LIN {X 103.742,Y 102.138,Z 83.038,A 180.000,B 0.000,C 180.000} C_DIS
LIN {X 103.836,Y 102.012,Z 83.035,A 180.000,B 0.000,C 180.000} C_DIS
LIN {X 103.928,Y 101.885,Z 83.032,A 180.000,B 0.000,C 180.000} C_DIS
LIN {X 104.017,Y 101.755,Z 83.030,A 180.000,B 0.000,C 180.000} C_DIS
LIN {X 104.184,Y 101.489,Z 83.025,A 180.000,B 0.000,C 180.000} C_DIS
LIN {X 104.341,Y 101.216,Z 83.021,A 180.000,B 0.000,C 180.000} C_DIS
LIN {X 104.489,Y 100.938,Z 83.017,A 180.000,B 0.000,C 180.000} C_DIS
LIN {X 104.623,Y 100.654,Z 83.013,A 180.000,B 0.000,C 180.000} C_DIS
LIN {X 104.744,Y 100.363,Z 83.010,A 180.000,B 0.000,C 180.000} C_DIS
LIN {X 104.858,Y 100.069,Z 83.007,A 180.000,B 0.000,C 180.000} C_DIS
LIN {X 104.957,Y 99.770,Z 83.005,A 180.000,B 0.000,C 180.000} C_DIS
LIN {X 105.040,Y 99.466,Z 83.003,A 180.000,B 0.000,C 180.000} C_DIS
LIN {X 105.117,Y 99.161,Z 83.001,A 180.000,B 0.000,C 180.000} C_DIS
LIN {X 105.179,Y 98.852,Z 83.000,A 180.000,B 0.000,C 180.000} C_DIS
LIN {X 105.224,Y 98.540,Z 83.000,A 180.000,B 0.000,C 180.000} C_DIS
LIN {X 105.239,Y 98.417,Z 83.000,A 180.000,B 0.000,C 180.000} C_DIS
; Cutting Move Starts
LIN {X 105.250,Y 98.327,Z 83.000,A 180.000,B 0.000,C 180.000} C_DIS
LIN {X 105.268,Y 98.148,Z 83.000,A 180.000,B 0.000,C 180.000} C_DIS
LIN {X 105.282,Y 97.969,Z 83.000,A 180.000,B 0.000,C 180.000} C_DIS
LIN {X 105.289,Y 97.790,Z 83.000,A 180.000,B 0.000,C 180.000} C_DIS
LIN {X 105.293,Y 97.612,Z 83.000,A 180.000,B 0.000,C 180.000} C_DIS
LIN {X 105.293,Y 97.433,Z 83.000,A 180.000,B 0.000,C 180.000} C_DIS
LIN {X 105.290,Y 97.254,Z 83.000,A 180.000,B 0.000,C 180.000} C_DIS
LIN {X 105.285,Y 97.075,Z 83.000,A 180.000,B 0.000,C 180.000} C_DIS
LIN {X 105.272,Y 96.897,Z 83.000,A 180.000,B 0.000,C 180.000} C_DIS
LIN {X 105.256,Y 96.718,Z 83.000,A 180.000,B 0.000,C 180.000} C_DIS
LIN {X 105.233,Y 96.539,Z 83.000,A 180.000,B 0.000,C 180.000} C_DIS
LIN {X 105.210,Y 96.360,Z 83.000,A 180.000,B 0.000,C 180.000} C_DIS
LIN {X 105.184,Y 96.181,Z 83.000,A 180.000,B 0.000,C 180.000} C_DIS
LIN {X 105.150,Y 96.003,Z 83.000,A 180.000,B 0.000,C 180.000} C_DIS
LIN {X 105.120,Y 95.853,Z 83.000,A 180.000,B 0.000,C 180.000} C_DIS
LIN {X 105.113,Y 95.824,Z 83.000,A 180.000,B 0.000,C 180.000} C_DIS
LIN {X 105.068,Y 95.645,Z 83.000,A 180.000,B 0.000,C 180.000} C_DIS
LIN {X 105.022,Y 95.466,Z 83.000,A 180.000,B 0.000,C 180.000} C_DIS
LIN {X 104.975,Y 95.288,Z 83.000,A 180.000,B 0.000,C 180.000} C_DIS
LIN {X 104.941,Y 95.177,Z 83.000,A 180.000,B 0.000,C 180.000} C_DIS
LIN {X 104.920,Y 95.109,Z 83.000,A 180.000,B 0.000,C 180.000} C_DIS
LIN {X 104.860,Y 94.930,Z 83.000,A 180.000,B 0.000,C 180.000} C_DIS
LIN {X 104.792,Y 94.751,Z 83.000,A 180.000,B 0.000,C 180.000} C_DIS
LIN {X 104.762,Y 94.674,Z 83.000,A 180.000,B 0.000,C 180.000} C_DIS
LIN {X 104.722,Y 94.573,Z 83.000,A 180.000,B 0.000,C 180.000} C_DIS
LIN {X 104.650,Y 94.394,Z 83.000,A 180.000,B 0.000,C 180.000} C_DIS
LIN {X 104.584,Y 94.246,Z 83.000,A 180.000,B 0.000,C 180.000} C_DIS
LIN {X 104.570,Y 94.215,Z 83.000,A 180.000,B 0.000,C 180.000} C_DIS
LIN {X 104.483,Y 94.036,Z 83.000,A 180.000,B 0.000,C 180.000} C_DIS
LIN {X 104.405,Y 93.885,Z 83.000,A 180.000,B 0.000,C 180.000} C_DIS
LIN {X 104.391,Y 93.857,Z 83.000,A 180.000,B 0.000,C 180.000} C_DIS
LIN {X 104.292,Y 93.679,Z 83.000,A 180.000,B 0.000,C 180.000} C_DIS
LIN {X 104.226,Y 93.561,Z 83.000,A 180.000,B 0.000,C 180.000} C_DIS
LIN {X 104.190,Y 93.500,Z 83.000,A 180.000,B 0.000,C 180.000} C_DIS
LIN {X 104.082,Y 93.321,Z 83.000,A 180.000,B 0.000,C 180.000} C_DIS
LIN {X 104.047,Y 93.269,Z 83.000,A 180.000,B 0.000,C 180.000} C_DIS
LIN {X 103.963,Y 93.142,Z 83.000,A 180.000,B 0.000,C 180.000} C_DIS
LIN {X 103.869,Y 93.008,Z 83.000,A 180.000,B 0.000,C 180.000} C_DIS
LIN {X 103.837,Y 92.964,Z 83.000,A 180.000,B 0.000,C 180.000} C_DIS
LIN {X 103.705,Y 92.785,Z 83.000,A 180.000,B 0.000,C 180.000} C_DIS
LIN {X 103.690,Y 92.764,Z 83.000,A 180.000,B 0.000,C 180.000} C_DIS
LIN {X 103.569,Y 92.606,Z 83.000,A 180.000,B 0.000,C 180.000} C_DIS
LIN {X 103.511,Y 92.536,Z 83.000,A 180.000,B 0.000,C 180.000} C_DIS
LIN {X 103.419,Y 92.427,Z 83.000,A 180.000,B 0.000,C 180.000} C_DIS
LIN {X 103.332,Y 92.328,Z 83.000,A 180.000,B 0.000,C 180.000} C_DIS
LIN {X 103.258,Y 92.249,Z 83.000,A 180.000,B 0.000,C 180.000} C_DIS
LIN {X 103.153,Y 92.138,Z 83.000,A 180.000,B 0.000,C 180.000} C_DIS
LIN {X 103.089,Y 92.070,Z 83.000,A 180.000,B 0.000,C 180.000} C_DIS
LIN {X 102.975,Y 91.950,Z 83.000,A 180.000,B 0.000,C 180.000} C_DIS
LIN {X 102.914,Y 91.891,Z 83.000,A 180.000,B 0.000,C 180.000} C_DIS
LIN {X 102.796,Y 91.779,Z 83.000,A 180.000,B 0.000,C 180.000} C_DIS
LIN {X 102.723,Y 91.712,Z 83.000,A 180.000,B 0.000,C 180.000} C_DIS
LIN {X 102.617,Y 91.622,Z 83.000,A 180.000,B 0.000,C 180.000} C_DIS
LIN {X 102.513,Y 91.533,Z 83.000,A 180.000,B 0.000,C 180.000} C_DIS
LIN {X 102.438,Y 91.472,Z 83.000,A 180.000,B 0.000,C 180.000} C_DIS
LIN {X 102.296,Y 91.355,Z 83.000,A 180.000,B 0.000,C 180.000} C_DIS
LIN {X 102.260,Y 91.326,Z 83.000,A 180.000,B 0.000,C 180.000} C_DIS
LIN {X 102.081,Y 91.192,Z 83.000,A 180.000,B 0.000,C 180.000} C_DIS
LIN {X 102.060,Y 91.176,Z 83.000,A 180.000,B 0.000,C 180.000} C_DIS
LIN {X 101.902,Y 91.068,Z 83.000,A 180.000,B 0.000,C 180.000} C_DIS
LIN {X 101.796,Y 90.997,Z 83.000,A 180.000,B 0.000,C 180.000} C_DIS
LIN {X 101.723,Y 90.950,Z 83.000,A 180.000,B 0.000,C 180.000} C_DIS
LIN {X 101.545,Y 90.837,Z 83.000,A 180.000,B 0.000,C 180.000} C_DIS
LIN {X 101.514,Y 90.818,Z 83.000,A 180.000,B 0.000,C 180.000} C_DIS
LIN {X 101.366,Y 90.731,Z 83.000,A 180.000,B 0.000,C 180.000} C_DIS
LIN {X 101.203,Y 90.640,Z 83.000,A 180.000,B 0.000,C 180.000} C_DIS
LIN {X 101.187,Y 90.631,Z 83.000,A 180.000,B 0.000,C 180.000} C_DIS
LIN {X 101.008,Y 90.539,Z 83.000,A 180.000,B 0.000,C 180.000} C_DIS
LIN {X 100.844,Y 90.461,Z 83.000,A 180.000,B 0.000,C 180.000} C_DIS
LIN {X 100.829,Y 90.454,Z 83.000,A 180.000,B 0.000,C 180.000} C_DIS
LIN {X 100.651,Y 90.372,Z 83.000,A 180.000,B 0.000,C 180.000} C_DIS
LIN {X 100.472,Y 90.292,Z 83.000,A 180.000,B 0.000,C 180.000} C_DIS
LIN {X 100.447,Y 90.282,Z 83.000,A 180.000,B 0.000,C 180.000} C_DIS
LIN {X 100.293,Y 90.222,Z 83.000,A 180.000,B 0.000,C 180.000} C_DIS
LIN {X 100.114,Y 90.156,Z 83.000,A 180.000,B 0.000,C 180.000} C_DIS
LIN {X 99.951,Y 90.103,Z 83.000,A 180.000,B 0.000,C 180.000} C_DIS
LIN {X 99.936,Y 90.098,Z 83.000,A 180.000,B 0.000,C 180.000} C_DIS
LIN {X 99.757,Y 90.041,Z 83.000,A 180.000,B 0.000,C 180.000} C_DIS
LIN {X 99.578,Y 89.986,Z 83.000,A 180.000,B 0.000,C 180.000} C_DIS
LIN {X 99.399,Y 89.939,Z 83.000,A 180.000,B 0.000,C 180.000} C_DIS
LIN {X 99.341,Y 89.925,Z 83.000,A 180.000,B 0.000,C 180.000} C_DIS
LIN {X 99.221,Y 89.897,Z 83.000,A 180.000,B 0.000,C 180.000} C_DIS
LIN {X 99.042,Y 89.861,Z 83.000,A 180.000,B 0.000,C 180.000} C_DIS
LIN {X 98.863,Y 89.827,Z 83.000,A 180.000,B 0.000,C 180.000} C_DIS
LIN {X 98.684,Y 89.795,Z 83.000,A 180.000,B 0.000,C 180.000} C_DIS
LIN {X 98.505,Y 89.770,Z 83.000,A 180.000,B 0.000,C 180.000} C_DIS
LIN {X 98.327,Y 89.748,Z 83.000,A 180.000,B 0.000,C 180.000} C_DIS
LIN {X 98.148,Y 89.733,Z 83.000,A 180.000,B 0.000,C 180.000} C_DIS
LIN {X 97.969,Y 89.721,Z 83.000,A 180.000,B 0.000,C 180.000} C_DIS
LIN {X 97.790,Y 89.711,Z 83.000,A 180.000,B 0.000,C 180.000} C_DIS
LIN {X 97.612,Y 89.705,Z 83.000,A 180.000,B 0.000,C 180.000} C_DIS
LIN {X 97.433,Y 89.704,Z 83.000,A 180.000,B 0.000,C 180.000} C_DIS
LIN {X 97.254,Y 89.709,Z 83.000,A 180.000,B 0.000,C 180.000} C_DIS
LIN {X 97.075,Y 89.718,Z 83.000,A 180.000,B 0.000,C 180.000} C_DIS
LIN {X 96.897,Y 89.730,Z 83.000,A 180.000,B 0.000,C 180.000} C_DIS
LIN {X 96.718,Y 89.745,Z 83.000,A 180.000,B 0.000,C 180.000} C_DIS
LIN {X 96.704,Y 89.746,Z 83.000,A 180.000,B 0.000,C 180.000} C_DIS
LIN {X 96.539,Y 89.763,Z 83.000,A 180.000,B 0.000,C 180.000} C_DIS
LIN {X 96.360,Y 89.789,Z 83.000,A 180.000,B 0.000,C 180.000} C_DIS
LIN {X 96.181,Y 89.819,Z 83.000,A 180.000,B 0.000,C 180.000} C_DIS
LIN {X 96.003,Y 89.853,Z 83.000,A 180.000,B 0.000,C 180.000} C_DIS
LIN {X 95.824,Y 89.888,Z 83.000,A 180.000,B 0.000,C 180.000} C_DIS
LIN {X 95.659,Y 89.925,Z 83.000,A 180.000,B 0.000,C 180.000} C_DIS
LIN {X 95.645,Y 89.928,Z 83.000,A 180.000,B 0.000,C 180.000} C_DIS
LIN {X 95.466,Y 89.974,Z 83.000,A 180.000,B 0.000,C 180.000} C_DIS
LIN {X 95.288,Y 90.027,Z 83.000,A 180.000,B 0.000,C 180.000} C_DIS
LIN {X 95.109,Y 90.084,Z 83.000,A 180.000,B 0.000,C 180.000} C_DIS
LIN {X 94.930,Y 90.142,Z 83.000,A 180.000,B 0.000,C 180.000} C_DIS
LIN {X 94.751,Y 90.205,Z 83.000,A 180.000,B 0.000,C 180.000} C_DIS
LIN {X 94.573,Y 90.274,Z 83.000,A 180.000,B 0.000,C 180.000} C_DIS
LIN {X 94.553,Y 90.282,Z 83.000,A 180.000,B 0.000,C 180.000} C_DIS
LIN {X 94.394,Y 90.352,Z 83.000,A 180.000,B 0.000,C 180.000} C_DIS
LIN {X 94.215,Y 90.433,Z 83.000,A 180.000,B 0.000,C 180.000} C_DIS
LIN {X 94.156,Y 90.461,Z 83.000,A 180.000,B 0.000,C 180.000} C_DIS
LIN {X 94.036,Y 90.517,Z 83.000,A 180.000,B 0.000,C 180.000} C_DIS
LIN {X 93.857,Y 90.608,Z 83.000,A 180.000,B 0.000,C 180.000} C_DIS
LIN {X 93.797,Y 90.640,Z 83.000,A 180.000,B 0.000,C 180.000} C_DIS
LIN {X 93.679,Y 90.705,Z 83.000,A 180.000,B 0.000,C 180.000} C_DIS
LIN {X 93.500,Y 90.810,Z 83.000,A 180.000,B 0.000,C 180.000} C_DIS
LIN {X 93.486,Y 90.818,Z 83.000,A 180.000,B 0.000,C 180.000} C_DIS
LIN {X 93.321,Y 90.922,Z 83.000,A 180.000,B 0.000,C 180.000} C_DIS
LIN {X 93.204,Y 90.997,Z 83.000,A 180.000,B 0.000,C 180.000} C_DIS
LIN {X 93.142,Y 91.038,Z 83.000,A 180.000,B 0.000,C 180.000} C_DIS
LIN {X 92.964,Y 91.159,Z 83.000,A 180.000,B 0.000,C 180.000} C_DIS
LIN {X 92.940,Y 91.176,Z 83.000,A 180.000,B 0.000,C 180.000} C_DIS
LIN {X 92.785,Y 91.293,Z 83.000,A 180.000,B 0.000,C 180.000} C_DIS
LIN {X 92.704,Y 91.355,Z 83.000,A 180.000,B 0.000,C 180.000} C_DIS
LIN {X 92.606,Y 91.435,Z 83.000,A 180.000,B 0.000,C 180.000} C_DIS
LIN {X 92.487,Y 91.533,Z 83.000,A 180.000,B 0.000,C 180.000} C_DIS
LIN {X 92.427,Y 91.584,Z 83.000,A 180.000,B 0.000,C 180.000} C_DIS
LIN {X 92.277,Y 91.712,Z 83.000,A 180.000,B 0.000,C 180.000} C_DIS
LIN {X 92.249,Y 91.738,Z 83.000,A 180.000,B 0.000,C 180.000} C_DIS
LIN {X 92.086,Y 91.891,Z 83.000,A 180.000,B 0.000,C 180.000} C_DIS
LIN {X 92.070,Y 91.906,Z 83.000,A 180.000,B 0.000,C 180.000} C_DIS
LIN {X 91.911,Y 92.070,Z 83.000,A 180.000,B 0.000,C 180.000} C_DIS
LIN {X 91.891,Y 92.091,Z 83.000,A 180.000,B 0.000,C 180.000} C_DIS
LIN {X 91.742,Y 92.249,Z 83.000,A 180.000,B 0.000,C 180.000} C_DIS
LIN {X 91.712,Y 92.281,Z 83.000,A 180.000,B 0.000,C 180.000} C_DIS
LIN {X 91.581,Y 92.427,Z 83.000,A 180.000,B 0.000,C 180.000} C_DIS
LIN {X 91.533,Y 92.483,Z 83.000,A 180.000,B 0.000,C 180.000} C_DIS
LIN {X 91.431,Y 92.606,Z 83.000,A 180.000,B 0.000,C 180.000} C_DIS
LIN {X 91.355,Y 92.705,Z 83.000,A 180.000,B 0.000,C 180.000} C_DIS
LIN {X 91.295,Y 92.785,Z 83.000,A 180.000,B 0.000,C 180.000} C_DIS
LIN {X 91.176,Y 92.946,Z 83.000,A 180.000,B 0.000,C 180.000} C_DIS
LIN {X 91.163,Y 92.964,Z 83.000,A 180.000,B 0.000,C 180.000} C_DIS
LIN {X 91.037,Y 93.142,Z 83.000,A 180.000,B 0.000,C 180.000} C_DIS
LIN {X 90.997,Y 93.202,Z 83.000,A 180.000,B 0.000,C 180.000} C_DIS
LIN {X 90.918,Y 93.321,Z 83.000,A 180.000,B 0.000,C 180.000} C_DIS
LIN {X 90.818,Y 93.486,Z 83.000,A 180.000,B 0.000,C 180.000} C_DIS
LIN {X 90.810,Y 93.500,Z 83.000,A 180.000,B 0.000,C 180.000} C_DIS
LIN {X 90.708,Y 93.679,Z 83.000,A 180.000,B 0.000,C 180.000} C_DIS
LIN {X 90.640,Y 93.802,Z 83.000,A 180.000,B 0.000,C 180.000} C_DIS
LIN {X 90.609,Y 93.857,Z 83.000,A 180.000,B 0.000,C 180.000} C_DIS
LIN {X 90.517,Y 94.036,Z 83.000,A 180.000,B 0.000,C 180.000} C_DIS
LIN {X 90.461,Y 94.148,Z 83.000,A 180.000,B 0.000,C 180.000} C_DIS
LIN {X 90.430,Y 94.215,Z 83.000,A 180.000,B 0.000,C 180.000} C_DIS
LIN {X 90.350,Y 94.394,Z 83.000,A 180.000,B 0.000,C 180.000} C_DIS
LIN {X 90.282,Y 94.562,Z 83.000,A 180.000,B 0.000,C 180.000} C_DIS
LIN {X 90.278,Y 94.573,Z 83.000,A 180.000,B 0.000,C 180.000} C_DIS
LIN {X 90.208,Y 94.751,Z 83.000,A 180.000,B 0.000,C 180.000} C_DIS
LIN {X 90.140,Y 94.930,Z 83.000,A 180.000,B 0.000,C 180.000} C_DIS
LIN {X 90.103,Y 95.037,Z 83.000,A 180.000,B 0.000,C 180.000} C_DIS
LIN {X 90.080,Y 95.109,Z 83.000,A 180.000,B 0.000,C 180.000} C_DIS
LIN {X 90.025,Y 95.288,Z 83.000,A 180.000,B 0.000,C 180.000} C_DIS
LIN {X 89.978,Y 95.466,Z 83.000,A 180.000,B 0.000,C 180.000} C_DIS
LIN {X 89.932,Y 95.645,Z 83.000,A 180.000,B 0.000,C 180.000} C_DIS
LIN {X 89.925,Y 95.673,Z 83.000,A 180.000,B 0.000,C 180.000} C_DIS
LIN {X 89.887,Y 95.824,Z 83.000,A 180.000,B 0.000,C 180.000} C_DIS
LIN {X 89.850,Y 96.003,Z 83.000,A 180.000,B 0.000,C 180.000} C_DIS
LIN {X 89.816,Y 96.181,Z 83.000,A 180.000,B 0.000,C 180.000} C_DIS
LIN {X 89.790,Y 96.360,Z 83.000,A 180.000,B 0.000,C 180.000} C_DIS
LIN {X 89.767,Y 96.539,Z 83.000,A 180.000,B 0.000,C 180.000} C_DIS
LIN {X 89.756,Y 96.623,Z 83.000,A 180.000,B 0.000,C 180.000} C_DIS
LIN {X 89.746,Y 96.706,Z 83.000,A 180.000,B 0.000,C 180.000} C_DIS
LIN {X 89.744,Y 96.718,Z 83.000,A 180.000,B 0.000,C 180.000} C_DIS
LIN {X 89.728,Y 96.897,Z 83.000,A 180.000,B 0.000,C 180.000} C_DIS
LIN {X 89.715,Y 97.075,Z 83.000,A 180.000,B 0.000,C 180.000} C_DIS
LIN {X 89.710,Y 97.254,Z 83.000,A 180.000,B 0.000,C 180.000} C_DIS
LIN {X 89.707,Y 97.433,Z 83.000,A 180.000,B 0.000,C 180.000} C_DIS
LIN {X 89.707,Y 97.612,Z 83.000,A 180.000,B 0.000,C 180.000} C_DIS
LIN {X 89.711,Y 97.790,Z 83.000,A 180.000,B 0.000,C 180.000} C_DIS
LIN {X 89.718,Y 97.969,Z 83.000,A 180.000,B 0.000,C 180.000} C_DIS
LIN {X 89.732,Y 98.148,Z 83.000,A 180.000,B 0.000,C 180.000} C_DIS
LIN {X 89.746,Y 98.294,Z 83.000,A 180.000,B 0.000,C 180.000} C_DIS
LIN {X 89.750,Y 98.327,Z 83.000,A 180.000,B 0.000,C 180.000} C_DIS
LIN {X 89.772,Y 98.505,Z 83.000,A 180.000,B 0.000,C 180.000} C_DIS
LIN {X 89.797,Y 98.684,Z 83.000,A 180.000,B 0.000,C 180.000} C_DIS
LIN {X 89.824,Y 98.863,Z 83.000,A 180.000,B 0.000,C 180.000} C_DIS
LIN {X 89.859,Y 99.042,Z 83.000,A 180.000,B 0.000,C 180.000} C_DIS
LIN {X 89.897,Y 99.221,Z 83.000,A 180.000,B 0.000,C 180.000} C_DIS
LIN {X 89.925,Y 99.327,Z 83.000,A 180.000,B 0.000,C 180.000} C_DIS
LIN {X 89.943,Y 99.399,Z 83.000,A 180.000,B 0.000,C 180.000} C_DIS
LIN {X 89.989,Y 99.578,Z 83.000,A 180.000,B 0.000,C 180.000} C_DIS
LIN {X 90.038,Y 99.757,Z 83.000,A 180.000,B 0.000,C 180.000} C_DIS
LIN {X 90.095,Y 99.936,Z 83.000,A 180.000,B 0.000,C 180.000} C_DIS
LIN {X 90.103,Y 99.963,Z 83.000,A 180.000,B 0.000,C 180.000} C_DIS
LIN {X 90.157,Y 100.114,Z 83.000,A 180.000,B 0.000,C 180.000} C_DIS
LIN {X 90.225,Y 100.293,Z 83.000,A 180.000,B 0.000,C 180.000} C_DIS
LIN {X 90.282,Y 100.438,Z 83.000,A 180.000,B 0.000,C 180.000} C_DIS
LIN {X 90.295,Y 100.472,Z 83.000,A 180.000,B 0.000,C 180.000} C_DIS
LIN {X 90.370,Y 100.651,Z 83.000,A 180.000,B 0.000,C 180.000} C_DIS
LIN {X 90.450,Y 100.829,Z 83.000,A 180.000,B 0.000,C 180.000} C_DIS
LIN {X 90.461,Y 100.852,Z 83.000,A 180.000,B 0.000,C 180.000} C_DIS
LIN {X 90.540,Y 101.008,Z 83.000,A 180.000,B 0.000,C 180.000} C_DIS
LIN {X 90.634,Y 101.187,Z 83.000,A 180.000,B 0.000,C 180.000} C_DIS
LIN {X 90.732,Y 101.366,Z 83.000,A 180.000,B 0.000,C 180.000} C_DIS
LIN {X 90.818,Y 101.514,Z 83.000,A 180.000,B 0.000,C 180.000} C_DIS
LIN {X 90.836,Y 101.545,Z 83.000,A 180.000,B 0.000,C 180.000} C_DIS
LIN {X 90.947,Y 101.723,Z 83.000,A 180.000,B 0.000,C 180.000} C_DIS
LIN {X 90.997,Y 101.798,Z 83.000,A 180.000,B 0.000,C 180.000} C_DIS
LIN {X 91.067,Y 101.902,Z 83.000,A 180.000,B 0.000,C 180.000} C_DIS
LIN {X 91.176,Y 102.054,Z 83.000,A 180.000,B 0.000,C 180.000} C_DIS
LIN {X 91.196,Y 102.081,Z 83.000,A 180.000,B 0.000,C 180.000} C_DIS
LIN {X 91.328,Y 102.260,Z 83.000,A 180.000,B 0.000,C 180.000} C_DIS
LIN {X 91.355,Y 102.295,Z 83.000,A 180.000,B 0.000,C 180.000} C_DIS
LIN {X 91.467,Y 102.438,Z 83.000,A 180.000,B 0.000,C 180.000} C_DIS
LIN {X 91.533,Y 102.517,Z 83.000,A 180.000,B 0.000,C 180.000} C_DIS
LIN {X 91.619,Y 102.617,Z 83.000,A 180.000,B 0.000,C 180.000} C_DIS
LIN {X 91.712,Y 102.719,Z 83.000,A 180.000,B 0.000,C 180.000} C_DIS
LIN {X 91.784,Y 102.796,Z 83.000,A 180.000,B 0.000,C 180.000} C_DIS
LIN {X 91.891,Y 102.909,Z 83.000,A 180.000,B 0.000,C 180.000} C_DIS
LIN {X 91.953,Y 102.975,Z 83.000,A 180.000,B 0.000,C 180.000} C_DIS
LIN {X 92.070,Y 103.094,Z 83.000,A 180.000,B 0.000,C 180.000} C_DIS
LIN {X 92.133,Y 103.153,Z 83.000,A 180.000,B 0.000,C 180.000} C_DIS
LIN {X 92.249,Y 103.262,Z 83.000,A 180.000,B 0.000,C 180.000} C_DIS
LIN {X 92.328,Y 103.332,Z 83.000,A 180.000,B 0.000,C 180.000} C_DIS
LIN {X 92.427,Y 103.416,Z 83.000,A 180.000,B 0.000,C 180.000} C_DIS
LIN {X 92.541,Y 103.511,Z 83.000,A 180.000,B 0.000,C 180.000} C_DIS
LIN {X 92.606,Y 103.565,Z 83.000,A 180.000,B 0.000,C 180.000} C_DIS
LIN {X 92.762,Y 103.690,Z 83.000,A 180.000,B 0.000,C 180.000} C_DIS
LIN {X 92.785,Y 103.707,Z 83.000,A 180.000,B 0.000,C 180.000} C_DIS
LIN {X 92.964,Y 103.841,Z 83.000,A 180.000,B 0.000,C 180.000} C_DIS
LIN {X 93.003,Y 103.869,Z 83.000,A 180.000,B 0.000,C 180.000} C_DIS
LIN {X 93.142,Y 103.962,Z 83.000,A 180.000,B 0.000,C 180.000} C_DIS
LIN {X 93.273,Y 104.047,Z 83.000,A 180.000,B 0.000,C 180.000} C_DIS
LIN {X 93.321,Y 104.078,Z 83.000,A 180.000,B 0.000,C 180.000} C_DIS
LIN {X 93.500,Y 104.190,Z 83.000,A 180.000,B 0.000,C 180.000} C_DIS
LIN {X 93.561,Y 104.226,Z 83.000,A 180.000,B 0.000,C 180.000} C_DIS
LIN {X 93.679,Y 104.295,Z 83.000,A 180.000,B 0.000,C 180.000} C_DIS
LIN {X 93.857,Y 104.392,Z 83.000,A 180.000,B 0.000,C 180.000} C_DIS
LIN {X 93.883,Y 104.405,Z 83.000,A 180.000,B 0.000,C 180.000} C_DIS
LIN {X 94.036,Y 104.483,Z 83.000,A 180.000,B 0.000,C 180.000} C_DIS
LIN {X 94.215,Y 104.567,Z 83.000,A 180.000,B 0.000,C 180.000} C_DIS
LIN {X 94.251,Y 104.584,Z 83.000,A 180.000,B 0.000,C 180.000} C_DIS
LIN {X 94.394,Y 104.648,Z 83.000,A 180.000,B 0.000,C 180.000} C_DIS
LIN {X 94.573,Y 104.726,Z 83.000,A 180.000,B 0.000,C 180.000} C_DIS
LIN {X 94.667,Y 104.762,Z 83.000,A 180.000,B 0.000,C 180.000} C_DIS
LIN {X 94.751,Y 104.795,Z 83.000,A 180.000,B 0.000,C 180.000} C_DIS
LIN {X 94.930,Y 104.858,Z 83.000,A 180.000,B 0.000,C 180.000} C_DIS
LIN {X 95.109,Y 104.916,Z 83.000,A 180.000,B 0.000,C 180.000} C_DIS
LIN {X 95.186,Y 104.941,Z 83.000,A 180.000,B 0.000,C 180.000} C_DIS
LIN {X 95.288,Y 104.973,Z 83.000,A 180.000,B 0.000,C 180.000} C_DIS
LIN {X 95.466,Y 105.026,Z 83.000,A 180.000,B 0.000,C 180.000} C_DIS
LIN {X 95.645,Y 105.072,Z 83.000,A 180.000,B 0.000,C 180.000} C_DIS
LIN {X 95.824,Y 105.112,Z 83.000,A 180.000,B 0.000,C 180.000} C_DIS
LIN {X 95.865,Y 105.120,Z 83.000,A 180.000,B 0.000,C 180.000} C_DIS
LIN {X 96.003,Y 105.147,Z 83.000,A 180.000,B 0.000,C 180.000} C_DIS
LIN {X 96.181,Y 105.181,Z 83.000,A 180.000,B 0.000,C 180.000} C_DIS
LIN {X 96.360,Y 105.211,Z 83.000,A 180.000,B 0.000,C 180.000} C_DIS
LIN {X 96.539,Y 105.237,Z 83.000,A 180.000,B 0.000,C 180.000} C_DIS
LIN {X 96.718,Y 105.255,Z 83.000,A 180.000,B 0.000,C 180.000} C_DIS
LIN {X 96.897,Y 105.270,Z 83.000,A 180.000,B 0.000,C 180.000} C_DIS
LIN {X 97.075,Y 105.282,Z 83.000,A 180.000,B 0.000,C 180.000} C_DIS
LIN {X 97.254,Y 105.291,Z 83.000,A 180.000,B 0.000,C 180.000} C_DIS
LIN {X 97.433,Y 105.296,Z 83.000,A 180.000,B 0.000,C 180.000} C_DIS
LIN {X 97.612,Y 105.295,Z 83.000,A 180.000,B 0.000,C 180.000} C_DIS
LIN {X 97.790,Y 105.289,Z 83.000,A 180.000,B 0.000,C 180.000} C_DIS
LIN {X 97.969,Y 105.279,Z 83.000,A 180.000,B 0.000,C 180.000} C_DIS
LIN {X 98.148,Y 105.267,Z 83.000,A 180.000,B 0.000,C 180.000} C_DIS
LIN {X 98.327,Y 105.252,Z 83.000,A 180.000,B 0.000,C 180.000} C_DIS
LIN {X 98.505,Y 105.230,Z 83.000,A 180.000,B 0.000,C 180.000} C_DIS
LIN {X 98.684,Y 105.205,Z 83.000,A 180.000,B 0.000,C 180.000} C_DIS
LIN {X 98.863,Y 105.173,Z 83.000,A 180.000,B 0.000,C 180.000} C_DIS
LIN {X 99.042,Y 105.139,Z 83.000,A 180.000,B 0.000,C 180.000} C_DIS
LIN {X 99.135,Y 105.120,Z 83.000,A 180.000,B 0.000,C 180.000} C_DIS
LIN {X 99.221,Y 105.103,Z 83.000,A 180.000,B 0.000,C 180.000} C_DIS
LIN {X 99.399,Y 105.061,Z 83.000,A 180.000,B 0.000,C 180.000} C_DIS
LIN {X 99.578,Y 105.014,Z 83.000,A 180.000,B 0.000,C 180.000} C_DIS
LIN {X 99.757,Y 104.959,Z 83.000,A 180.000,B 0.000,C 180.000} C_DIS
LIN {X 99.814,Y 104.941,Z 83.000,A 180.000,B 0.000,C 180.000} C_DIS
LIN {X 99.936,Y 104.902,Z 83.000,A 180.000,B 0.000,C 180.000} C_DIS
LIN {X 100.114,Y 104.844,Z 83.000,A 180.000,B 0.000,C 180.000} C_DIS
LIN {X 100.293,Y 104.778,Z 83.000,A 180.000,B 0.000,C 180.000} C_DIS
LIN {X 100.333,Y 104.762,Z 83.000,A 180.000,B 0.000,C 180.000} C_DIS
LIN {X 100.472,Y 104.708,Z 83.000,A 180.000,B 0.000,C 180.000} C_DIS
LIN {X 100.651,Y 104.628,Z 83.000,A 180.000,B 0.000,C 180.000} C_DIS
LIN {X 100.749,Y 104.584,Z 83.000,A 180.000,B 0.000,C 180.000} C_DIS
LIN {X 100.829,Y 104.546,Z 83.000,A 180.000,B 0.000,C 180.000} C_DIS
LIN {X 101.008,Y 104.461,Z 83.000,A 180.000,B 0.000,C 180.000} C_DIS
LIN {X 101.117,Y 104.405,Z 83.000,A 180.000,B 0.000,C 180.000} C_DIS
LIN {X 101.187,Y 104.369,Z 83.000,A 180.000,B 0.000,C 180.000} C_DIS
LIN {X 101.366,Y 104.269,Z 83.000,A 180.000,B 0.000,C 180.000} C_DIS
LIN {X 101.439,Y 104.226,Z 83.000,A 180.000,B 0.000,C 180.000} C_DIS
LIN {X 101.545,Y 104.163,Z 83.000,A 180.000,B 0.000,C 180.000} C_DIS
LIN {X 101.727,Y 104.047,Z 83.000,A 180.000,B 0.000,C 180.000} C_DIS
LIN {X 101.902,Y 103.932,Z 83.000,A 180.000,B 0.000,C 180.000} C_DIS
LIN {X 101.997,Y 103.869,Z 83.000,A 180.000,B 0.000,C 180.000} C_DIS
LIN {X 102.081,Y 103.808,Z 83.000,A 180.000,B 0.000,C 180.000} C_DIS
LIN {X 102.238,Y 103.690,Z 83.000,A 180.000,B 0.000,C 180.000} C_DIS
LIN {X 102.260,Y 103.674,Z 83.000,A 180.000,B 0.000,C 180.000} C_DIS
LIN {X 102.438,Y 103.528,Z 83.000,A 180.000,B 0.000,C 180.000} C_DIS
LIN {X 102.459,Y 103.511,Z 83.000,A 180.000,B 0.000,C 180.000} C_DIS
LIN {X 102.617,Y 103.378,Z 83.000,A 180.000,B 0.000,C 180.000} C_DIS
LIN {X 102.672,Y 103.332,Z 83.000,A 180.000,B 0.000,C 180.000} C_DIS
LIN {X 102.796,Y 103.221,Z 83.000,A 180.000,B 0.000,C 180.000} C_DIS
LIN {X 102.867,Y 103.153,Z 83.000,A 180.000,B 0.000,C 180.000} C_DIS
LIN {X 102.975,Y 103.050,Z 83.000,A 180.000,B 0.000,C 180.000} C_DIS
LIN {X 103.047,Y 102.975,Z 83.000,A 180.000,B 0.000,C 180.000} C_DIS
LIN {X 103.153,Y 102.862,Z 83.000,A 180.000,B 0.000,C 180.000} C_DIS
LIN {X 103.216,Y 102.796,Z 83.000,A 180.000,B 0.000,C 180.000} C_DIS
LIN {X 103.332,Y 102.672,Z 83.000,A 180.000,B 0.000,C 180.000} C_DIS
LIN {X 103.381,Y 102.617,Z 83.000,A 180.000,B 0.000,C 180.000} C_DIS
LIN {X 103.511,Y 102.464,Z 83.000,A 180.000,B 0.000,C 180.000} C_DIS
LIN {X 103.533,Y 102.438,Z 83.000,A 180.000,B 0.000,C 180.000} C_DIS
LIN {X 103.672,Y 102.260,Z 83.000,A 180.000,B 0.000,C 180.000} C_DIS
LIN {X 103.690,Y 102.236,Z 83.000,A 180.000,B 0.000,C 180.000} C_DIS
LIN {X 103.804,Y 102.081,Z 83.000,A 180.000,B 0.000,C 180.000} C_DIS
LIN {X 103.869,Y 101.992,Z 83.000,A 180.000,B 0.000,C 180.000} C_DIS
LIN {X 103.933,Y 101.902,Z 83.000,A 180.000,B 0.000,C 180.000} C_DIS
LIN {X 104.047,Y 101.731,Z 83.000,A 180.000,B 0.000,C 180.000} C_DIS
LIN {X 104.053,Y 101.723,Z 83.000,A 180.000,B 0.000,C 180.000} C_DIS
LIN {X 104.164,Y 101.545,Z 83.000,A 180.000,B 0.000,C 180.000} C_DIS
LIN {X 104.226,Y 101.439,Z 83.000,A 180.000,B 0.000,C 180.000} C_DIS
LIN {X 104.268,Y 101.366,Z 83.000,A 180.000,B 0.000,C 180.000} C_DIS
LIN {X 104.366,Y 101.187,Z 83.000,A 180.000,B 0.000,C 180.000} C_DIS
LIN {X 104.405,Y 101.115,Z 83.000,A 180.000,B 0.000,C 180.000} C_DIS
LIN {X 104.460,Y 101.008,Z 83.000,A 180.000,B 0.000,C 180.000} C_DIS
LIN {X 104.550,Y 100.829,Z 83.000,A 180.000,B 0.000,C 180.000} C_DIS
LIN {X 104.584,Y 100.754,Z 83.000,A 180.000,B 0.000,C 180.000} C_DIS
LIN {X 104.630,Y 100.651,Z 83.000,A 180.000,B 0.000,C 180.000} C_DIS
LIN {X 104.705,Y 100.472,Z 83.000,A 180.000,B 0.000,C 180.000} C_DIS
LIN {X 104.762,Y 100.326,Z 83.000,A 180.000,B 0.000,C 180.000} C_DIS
LIN {X 104.775,Y 100.293,Z 83.000,A 180.000,B 0.000,C 180.000} C_DIS
LIN {X 104.843,Y 100.114,Z 83.000,A 180.000,B 0.000,C 180.000} C_DIS
LIN {X 104.905,Y 99.936,Z 83.000,A 180.000,B 0.000,C 180.000} C_DIS
LIN {X 104.941,Y 99.823,Z 83.000,A 180.000,B 0.000,C 180.000} C_DIS
LIN {X 104.962,Y 99.757,Z 83.000,A 180.000,B 0.000,C 180.000} C_DIS
LIN {X 105.011,Y 99.578,Z 83.000,A 180.000,B 0.000,C 180.000} C_DIS
LIN {X 105.057,Y 99.399,Z 83.000,A 180.000,B 0.000,C 180.000} C_DIS
LIN {X 105.103,Y 99.221,Z 83.000,A 180.000,B 0.000,C 180.000} C_DIS
LIN {X 105.120,Y 99.147,Z 83.000,A 180.000,B 0.000,C 180.000} C_DIS
LIN {X 105.141,Y 99.042,Z 83.000,A 180.000,B 0.000,C 180.000} C_DIS
LIN {X 105.176,Y 98.863,Z 83.000,A 180.000,B 0.000,C 180.000} C_DIS
LIN {X 105.203,Y 98.684,Z 83.000,A 180.000,B 0.000,C 180.000} C_DIS
LIN {X 105.228,Y 98.505,Z 83.000,A 180.000,B 0.000,C 180.000} C_DIS
LIN {X 105.239,Y 98.417,Z 83.000,A 180.000,B 0.000,C 180.000} C_DIS
; Link Move Starts
LIN {X 105.272,Y 98.120,Z 83.000,A 180.000,B 0.000,C 180.000} C_DIS
LIN {X 105.290,Y 97.831,Z 82.999,A 180.000,B 0.000,C 180.000} C_DIS
LIN {X 105.295,Y 97.531,Z 82.998,A 180.000,B 0.000,C 180.000} C_DIS
LIN {X 105.292,Y 97.230,Z 82.997,A 180.000,B 0.000,C 180.000} C_DIS
LIN {X 105.278,Y 96.934,Z 82.995,A 180.000,B 0.000,C 180.000} C_DIS
LIN {X 105.251,Y 96.642,Z 82.992,A 180.000,B 0.000,C 180.000} C_DIS
LIN {X 105.213,Y 96.341,Z 82.990,A 180.000,B 0.000,C 180.000} C_DIS
LIN {X 105.168,Y 96.055,Z 82.987,A 180.000,B 0.000,C 180.000} C_DIS
LIN {X 105.107,Y 95.757,Z 82.983,A 180.000,B 0.000,C 180.000} C_DIS
LIN {X 105.034,Y 95.466,Z 82.979,A 180.000,B 0.000,C 180.000} C_DIS
LIN {X 104.958,Y 95.187,Z 82.975,A 180.000,B 0.000,C 180.000} C_DIS
LIN {X 104.869,Y 94.911,Z 82.970,A 180.000,B 0.000,C 180.000} C_DIS
LIN {X 104.815,Y 94.765,Z 82.968,A 180.000,B 0.000,C 180.000} C_DIS
LIN {X 104.760,Y 94.620,Z 82.965,A 180.000,B 0.000,C 180.000} C_DIS
LIN {X 104.707,Y 94.483,Z 82.963,A 180.000,B 0.000,C 180.000} C_DIS
LIN {X 104.651,Y 94.347,Z 82.960,A 180.000,B 0.000,C 180.000} C_DIS
LIN {X 104.592,Y 94.213,Z 82.957,A 180.000,B 0.000,C 180.000} C_DIS
LIN {X 104.531,Y 94.079,Z 82.954,A 180.000,B 0.000,C 180.000} C_DIS
LIN {X 104.462,Y 93.943,Z 82.951,A 180.000,B 0.000,C 180.000} C_DIS
LIN {X 104.392,Y 93.808,Z 82.948,A 180.000,B 0.000,C 180.000} C_DIS
LIN {X 104.320,Y 93.674,Z 82.945,A 180.000,B 0.000,C 180.000} C_DIS
LIN {X 104.247,Y 93.541,Z 82.942,A 180.000,B 0.000,C 180.000} C_DIS
LIN {X 104.174,Y 93.415,Z 82.939,A 180.000,B 0.000,C 180.000} C_DIS
LIN {X 104.100,Y 93.291,Z 82.935,A 180.000,B 0.000,C 180.000} C_DIS
LIN {X 104.016,Y 93.163,Z 82.932,A 180.000,B 0.000,C 180.000} C_DIS
LIN {X 103.931,Y 93.035,Z 82.928,A 180.000,B 0.000,C 180.000} C_DIS
LIN {X 103.846,Y 92.915,Z 82.925,A 180.000,B 0.000,C 180.000} C_DIS
LIN {X 103.761,Y 92.795,Z 82.921,A 180.000,B 0.000,C 180.000} C_DIS
LIN {X 103.671,Y 92.673,Z 82.917,A 180.000,B 0.000,C 180.000} C_DIS
LIN {X 103.579,Y 92.552,Z 82.913,A 180.000,B 0.000,C 180.000} C_DIS
LIN {X 103.486,Y 92.440,Z 82.910,A 180.000,B 0.000,C 180.000} C_DIS
LIN {X 103.393,Y 92.328,Z 82.906,A 180.000,B 0.000,C 180.000} C_DIS
LIN {X 103.292,Y 92.216,Z 82.902,A 180.000,B 0.000,C 180.000} C_DIS
LIN {X 103.190,Y 92.105,Z 82.898,A 180.000,B 0.000,C 180.000} C_DIS
LIN {X 103.089,Y 91.996,Z 82.893,A 180.000,B 0.000,C 180.000} C_DIS
LIN {X 102.987,Y 91.888,Z 82.889,A 180.000,B 0.000,C 180.000} C_DIS
LIN {X 102.877,Y 91.781,Z 82.885,A 180.000,B 0.000,C 180.000} C_DIS
LIN {X 102.767,Y 91.675,Z 82.880,A 180.000,B 0.000,C 180.000} C_DIS
LIN {X 102.657,Y 91.578,Z 82.876,A 180.000,B 0.000,C 180.000} C_DIS
LIN {X 102.546,Y 91.481,Z 82.872,A 180.000,B 0.000,C 180.000} C_DIS
LIN {X 102.433,Y 91.385,Z 82.867,A 180.000,B 0.000,C 180.000} C_DIS
LIN {X 102.320,Y 91.290,Z 82.862,A 180.000,B 0.000,C 180.000} C_DIS
LIN {X 102.200,Y 91.197,Z 82.858,A 180.000,B 0.000,C 180.000} C_DIS
LIN {X 102.079,Y 91.104,Z 82.853,A 180.000,B 0.000,C 180.000} C_DIS
LIN {X 101.959,Y 91.019,Z 82.848,A 180.000,B 0.000,C 180.000} C_DIS
LIN {X 101.837,Y 90.935,Z 82.843,A 180.000,B 0.000,C 180.000} C_DIS
LIN {X 101.710,Y 90.851,Z 82.838,A 180.000,B 0.000,C 180.000} C_DIS
LIN {X 101.647,Y 90.810,Z 82.836,A 180.000,B 0.000,C 180.000} C_DIS
LIN {X 101.583,Y 90.768,Z 82.833,A 180.000,B 0.000,C 180.000} C_DIS
LIN {X 101.458,Y 90.691,Z 82.828,A 180.000,B 0.000,C 180.000} C_DIS
LIN {X 101.333,Y 90.615,Z 82.823,A 180.000,B 0.000,C 180.000} C_DIS
LIN {X 101.266,Y 90.577,Z 82.821,A 180.000,B 0.000,C 180.000} C_DIS
LIN {X 101.197,Y 90.540,Z 82.818,A 180.000,B 0.000,C 180.000} C_DIS
LIN {X 101.129,Y 90.503,Z 82.815,A 180.000,B 0.000,C 180.000} C_DIS
LIN {X 101.061,Y 90.467,Z 82.813,A 180.000,B 0.000,C 180.000} C_DIS
LIN {X 100.995,Y 90.433,Z 82.810,A 180.000,B 0.000,C 180.000} C_DIS
LIN {X 100.928,Y 90.400,Z 82.808,A 180.000,B 0.000,C 180.000} C_DIS
LIN {X 100.794,Y 90.334,Z 82.802,A 180.000,B 0.000,C 180.000} C_DIS
LIN {X 100.724,Y 90.301,Z 82.800,A 180.000,B 0.000,C 180.000} C_DIS
LIN {X 100.584,Y 90.235,Z 82.794,A 180.000,B 0.000,C 180.000} C_DIS
LIN {X 100.513,Y 90.203,Z 82.792,A 180.000,B 0.000,C 180.000} C_DIS
LIN {X 100.445,Y 90.174,Z 82.789,A 180.000,B 0.000,C 180.000} C_DIS
LIN {X 100.376,Y 90.146,Z 82.786,A 180.000,B 0.000,C 180.000} C_DIS
LIN {X 100.239,Y 90.091,Z 82.781,A 180.000,B 0.000,C 180.000} C_DIS
LIN {X 100.170,Y 90.065,Z 82.779,A 180.000,B 0.000,C 180.000} C_DIS
LIN {X 100.100,Y 90.041,Z 82.776,A 180.000,B 0.000,C 180.000} C_DIS
LIN {X 99.961,Y 89.993,Z 82.771,A 180.000,B 0.000,C 180.000} C_DIS
LIN {X 99.887,Y 89.968,Z 82.768,A 180.000,B 0.000,C 180.000} C_DIS
LIN {X 99.740,Y 89.918,Z 82.763,A 180.000,B 0.000,C 180.000} C_DIS
LIN {X 99.666,Y 89.894,Z 82.760,A 180.000,B 0.000,C 180.000} C_DIS
LIN {X 99.595,Y 89.872,Z 82.757,A 180.000,B 0.000,C 180.000} C_DIS
LIN {X 99.523,Y 89.852,Z 82.755,A 180.000,B 0.000,C 180.000} C_DIS
LIN {X 99.380,Y 89.813,Z 82.750,A 180.000,B 0.000,C 180.000} C_DIS
LIN {X 99.308,Y 89.794,Z 82.747,A 180.000,B 0.000,C 180.000} C_DIS
LIN {X 99.236,Y 89.777,Z 82.744,A 180.000,B 0.000,C 180.000} C_DIS
LIN {X 99.091,Y 89.746,Z 82.739,A 180.000,B 0.000,C 180.000} C_DIS
LIN {X 99.017,Y 89.730,Z 82.737,A 180.000,B 0.000,C 180.000} C_DIS
LIN {X 98.870,Y 89.700,Z 82.731,A 180.000,B 0.000,C 180.000} C_DIS
LIN {X 98.796,Y 89.684,Z 82.729,A 180.000,B 0.000,C 180.000} C_DIS
LIN {X 98.720,Y 89.670,Z 82.726,A 180.000,B 0.000,C 180.000} C_DIS
LIN {X 98.643,Y 89.658,Z 82.723,A 180.000,B 0.000,C 180.000} C_DIS
LIN {X 98.490,Y 89.633,Z 82.718,A 180.000,B 0.000,C 180.000} C_DIS
LIN {X 98.417,Y 89.623,Z 82.715,A 180.000,B 0.000,C 180.000} C_DIS
LIN {X 98.343,Y 89.614,Z 82.713,A 180.000,B 0.000,C 180.000} C_DIS
LIN {X 98.196,Y 89.599,Z 82.708,A 180.000,B 0.000,C 180.000} C_DIS
LIN {X 98.120,Y 89.592,Z 82.705,A 180.000,B 0.000,C 180.000} C_DIS
LIN {X 98.044,Y 89.585,Z 82.702,A 180.000,B 0.000,C 180.000} C_DIS
LIN {X 97.892,Y 89.573,Z 82.697,A 180.000,B 0.000,C 180.000} C_DIS
LIN {X 97.817,Y 89.568,Z 82.694,A 180.000,B 0.000,C 180.000} C_DIS
LIN {X 97.743,Y 89.564,Z 82.692,A 180.000,B 0.000,C 180.000} C_DIS
LIN {X 97.592,Y 89.558,Z 82.686,A 180.000,B 0.000,C 180.000} C_DIS
LIN {X 97.517,Y 89.555,Z 82.684,A 180.000,B 0.000,C 180.000} C_DIS
LIN {X 97.441,Y 89.554,Z 82.681,A 180.000,B 0.000,C 180.000} C_DIS
LIN {X 97.365,Y 89.555,Z 82.678,A 180.000,B 0.000,C 180.000} C_DIS
LIN {X 97.289,Y 89.556,Z 82.676,A 180.000,B 0.000,C 180.000} C_DIS
LIN {X 97.213,Y 89.557,Z 82.673,A 180.000,B 0.000,C 180.000} C_DIS
LIN {X 97.137,Y 89.559,Z 82.671,A 180.000,B 0.000,C 180.000} C_DIS
LIN {X 96.908,Y 89.570,Z 82.663,A 180.000,B 0.000,C 180.000} C_DIS
LIN {X 96.832,Y 89.575,Z 82.660,A 180.000,B 0.000,C 180.000} C_DIS
LIN {X 96.679,Y 89.585,Z 82.655,A 180.000,B 0.000,C 180.000} C_DIS
LIN {X 96.605,Y 89.591,Z 82.652,A 180.000,B 0.000,C 180.000} C_DIS
LIN {X 96.531,Y 89.598,Z 82.649,A 180.000,B 0.000,C 180.000} C_DIS
LIN {X 96.456,Y 89.607,Z 82.647,A 180.000,B 0.000,C 180.000} C_DIS
LIN {X 96.307,Y 89.626,Z 82.641,A 180.000,B 0.000,C 180.000} C_DIS
LIN {X 96.232,Y 89.637,Z 82.639,A 180.000,B 0.000,C 180.000} C_DIS
LIN {X 96.157,Y 89.649,Z 82.636,A 180.000,B 0.000,C 180.000} C_DIS
LIN {X 96.006,Y 89.676,Z 82.631,A 180.000,B 0.000,C 180.000} C_DIS
LIN {X 95.929,Y 89.689,Z 82.628,A 180.000,B 0.000,C 180.000} C_DIS
LIN {X 95.776,Y 89.717,Z 82.623,A 180.000,B 0.000,C 180.000} C_DIS
LIN {X 95.703,Y 89.731,Z 82.620,A 180.000,B 0.000,C 180.000} C_DIS
LIN {X 95.630,Y 89.747,Z 82.617,A 180.000,B 0.000,C 180.000} C_DIS
LIN {X 95.557,Y 89.764,Z 82.615,A 180.000,B 0.000,C 180.000} C_DIS
LIN {X 95.411,Y 89.799,Z 82.610,A 180.000,B 0.000,C 180.000} C_DIS
LIN {X 95.339,Y 89.818,Z 82.607,A 180.000,B 0.000,C 180.000} C_DIS
LIN {X 95.267,Y 89.838,Z 82.604,A 180.000,B 0.000,C 180.000} C_DIS
LIN {X 95.120,Y 89.883,Z 82.599,A 180.000,B 0.000,C 180.000} C_DIS
LIN {X 95.045,Y 89.905,Z 82.596,A 180.000,B 0.000,C 180.000} C_DIS
LIN {X 94.895,Y 89.951,Z 82.591,A 180.000,B 0.000,C 180.000} C_DIS
LIN {X 94.823,Y 89.973,Z 82.588,A 180.000,B 0.000,C 180.000} C_DIS
LIN {X 94.752,Y 89.997,Z 82.586,A 180.000,B 0.000,C 180.000} C_DIS
LIN {X 94.681,Y 90.023,Z 82.583,A 180.000,B 0.000,C 180.000} C_DIS
LIN {X 94.539,Y 90.074,Z 82.578,A 180.000,B 0.000,C 180.000} C_DIS
LIN {X 94.468,Y 90.101,Z 82.575,A 180.000,B 0.000,C 180.000} C_DIS
LIN {X 94.398,Y 90.130,Z 82.572,A 180.000,B 0.000,C 180.000} C_DIS
LIN {X 94.258,Y 90.190,Z 82.567,A 180.000,B 0.000,C 180.000} C_DIS
LIN {X 94.187,Y 90.220,Z 82.564,A 180.000,B 0.000,C 180.000} C_DIS
LIN {X 94.117,Y 90.252,Z 82.562,A 180.000,B 0.000,C 180.000} C_DIS
LIN {X 93.978,Y 90.315,Z 82.556,A 180.000,B 0.000,C 180.000} C_DIS
LIN {X 93.909,Y 90.346,Z 82.554,A 180.000,B 0.000,C 180.000} C_DIS
LIN {X 93.841,Y 90.380,Z 82.551,A 180.000,B 0.000,C 180.000} C_DIS
LIN {X 93.705,Y 90.447,Z 82.546,A 180.000,B 0.000,C 180.000} C_DIS
LIN {X 93.638,Y 90.482,Z 82.543,A 180.000,B 0.000,C 180.000} C_DIS
LIN {X 93.571,Y 90.518,Z 82.540,A 180.000,B 0.000,C 180.000} C_DIS
LIN {X 93.439,Y 90.593,Z 82.535,A 180.000,B 0.000,C 180.000} C_DIS
LIN {X 93.372,Y 90.631,Z 82.532,A 180.000,B 0.000,C 180.000} C_DIS
LIN {X 93.306,Y 90.670,Z 82.530,A 180.000,B 0.000,C 180.000} C_DIS
LIN {X 93.175,Y 90.751,Z 82.524,A 180.000,B 0.000,C 180.000} C_DIS
LIN {X 93.109,Y 90.791,Z 82.522,A 180.000,B 0.000,C 180.000} C_DIS
LIN {X 93.044,Y 90.833,Z 82.519,A 180.000,B 0.000,C 180.000} C_DIS
LIN {X 92.916,Y 90.916,Z 82.514,A 180.000,B 0.000,C 180.000} C_DIS
LIN {X 92.853,Y 90.957,Z 82.511,A 180.000,B 0.000,C 180.000} C_DIS
LIN {X 92.791,Y 91.000,Z 82.508,A 180.000,B 0.000,C 180.000} C_DIS
LIN {X 92.730,Y 91.044,Z 82.506,A 180.000,B 0.000,C 180.000} C_DIS
LIN {X 92.607,Y 91.134,Z 82.500,A 180.000,B 0.000,C 180.000} C_DIS
LIN {X 92.546,Y 91.180,Z 82.498,A 180.000,B 0.000,C 180.000} C_DIS
LIN {X 92.486,Y 91.227,Z 82.495,A 180.000,B 0.000,C 180.000} C_DIS
LIN {X 92.364,Y 91.325,Z 82.490,A 180.000,B 0.000,C 180.000} C_DIS
LIN {X 92.303,Y 91.374,Z 82.487,A 180.000,B 0.000,C 180.000} C_DIS
LIN {X 92.184,Y 91.471,Z 82.482,A 180.000,B 0.000,C 180.000} C_DIS
LIN {X 92.126,Y 91.520,Z 82.479,A 180.000,B 0.000,C 180.000} C_DIS
LIN {X 92.069,Y 91.569,Z 82.476,A 180.000,B 0.000,C 180.000} C_DIS
LIN {X 92.013,Y 91.621,Z 82.474,A 180.000,B 0.000,C 180.000} C_DIS
LIN {X 91.901,Y 91.724,Z 82.468,A 180.000,B 0.000,C 180.000} C_DIS
LIN {X 91.845,Y 91.776,Z 82.466,A 180.000,B 0.000,C 180.000} C_DIS
LIN {X 91.791,Y 91.830,Z 82.463,A 180.000,B 0.000,C 180.000} C_DIS
LIN {X 91.682,Y 91.942,Z 82.458,A 180.000,B 0.000,C 180.000} C_DIS
LIN {X 91.628,Y 91.997,Z 82.455,A 180.000,B 0.000,C 180.000} C_DIS
LIN {X 91.521,Y 92.108,Z 82.449,A 180.000,B 0.000,C 180.000} C_DIS
LIN {X 91.468,Y 92.163,Z 82.447,A 180.000,B 0.000,C 180.000} C_DIS
LIN {X 91.416,Y 92.219,Z 82.444,A 180.000,B 0.000,C 180.000} C_DIS
LIN {X 91.366,Y 92.276,Z 82.441,A 180.000,B 0.000,C 180.000} C_DIS
LIN {X 91.265,Y 92.393,Z 82.436,A 180.000,B 0.000,C 180.000} C_DIS
LIN {X 91.215,Y 92.451,Z 82.433,A 180.000,B 0.000,C 180.000} C_DIS
LIN {X 91.166,Y 92.512,Z 82.431,A 180.000,B 0.000,C 180.000} C_DIS
LIN {X 91.072,Y 92.633,Z 82.425,A 180.000,B 0.000,C 180.000} C_DIS
LIN {X 91.026,Y 92.693,Z 82.423,A 180.000,B 0.000,C 180.000} C_DIS
LIN {X 90.980,Y 92.754,Z 82.420,A 180.000,B 0.000,C 180.000} C_DIS
LIN {X 90.887,Y 92.877,Z 82.415,A 180.000,B 0.000,C 180.000} C_DIS
LIN {X 90.842,Y 92.940,Z 82.412,A 180.000,B 0.000,C 180.000} C_DIS
LIN {X 90.798,Y 93.003,Z 82.409,A 180.000,B 0.000,C 180.000} C_DIS
LIN {X 90.711,Y 93.128,Z 82.404,A 180.000,B 0.000,C 180.000} C_DIS
LIN {X 90.668,Y 93.191,Z 82.401,A 180.000,B 0.000,C 180.000} C_DIS
LIN {X 90.628,Y 93.255,Z 82.399,A 180.000,B 0.000,C 180.000} C_DIS
LIN {X 90.546,Y 93.388,Z 82.393,A 180.000,B 0.000,C 180.000} C_DIS
LIN {X 90.506,Y 93.455,Z 82.390,A 180.000,B 0.000,C 180.000} C_DIS
LIN {X 90.467,Y 93.522,Z 82.388,A 180.000,B 0.000,C 180.000} C_DIS
LIN {X 90.390,Y 93.656,Z 82.382,A 180.000,B 0.000,C 180.000} C_DIS
LIN {X 90.352,Y 93.723,Z 82.380,A 180.000,B 0.000,C 180.000} C_DIS
LIN {X 90.315,Y 93.790,Z 82.377,A 180.000,B 0.000,C 180.000} C_DIS
LIN {X 90.242,Y 93.927,Z 82.372,A 180.000,B 0.000,C 180.000} C_DIS
LIN {X 90.206,Y 93.995,Z 82.369,A 180.000,B 0.000,C 180.000} C_DIS
LIN {X 90.173,Y 94.065,Z 82.366,A 180.000,B 0.000,C 180.000} C_DIS
LIN {X 90.108,Y 94.203,Z 82.361,A 180.000,B 0.000,C 180.000} C_DIS
LIN {X 90.076,Y 94.272,Z 82.358,A 180.000,B 0.000,C 180.000} C_DIS
LIN {X 90.045,Y 94.342,Z 82.355,A 180.000,B 0.000,C 180.000} C_DIS
LIN {X 90.015,Y 94.414,Z 82.353,A 180.000,B 0.000,C 180.000} C_DIS
LIN {X 89.955,Y 94.558,Z 82.347,A 180.000,B 0.000,C 180.000} C_DIS
LIN {X 89.926,Y 94.631,Z 82.345,A 180.000,B 0.000,C 180.000} C_DIS
LIN {X 89.868,Y 94.774,Z 82.339,A 180.000,B 0.000,C 180.000} C_DIS
LIN {X 89.840,Y 94.845,Z 82.337,A 180.000,B 0.000,C 180.000} C_DIS
LIN {X 89.814,Y 94.918,Z 82.334,A 180.000,B 0.000,C 180.000} C_DIS
LIN {X 89.765,Y 95.064,Z 82.328,A 180.000,B 0.000,C 180.000} C_DIS
LIN {X 89.740,Y 95.137,Z 82.326,A 180.000,B 0.000,C 180.000} C_DIS
LIN {X 89.717,Y 95.211,Z 82.323,A 180.000,B 0.000,C 180.000} C_DIS
LIN {X 89.696,Y 95.286,Z 82.320,A 180.000,B 0.000,C 180.000} C_DIS
LIN {X 89.655,Y 95.435,Z 82.315,A 180.000,B 0.000,C 180.000} C_DIS
LIN {X 89.634,Y 95.510,Z 82.312,A 180.000,B 0.000,C 180.000} C_DIS
LIN {X 89.593,Y 95.660,Z 82.307,A 180.000,B 0.000,C 180.000} C_DIS
LIN {X 89.573,Y 95.735,Z 82.304,A 180.000,B 0.000,C 180.000} C_DIS
LIN {X 89.555,Y 95.810,Z 82.301,A 180.000,B 0.000,C 180.000} C_DIS
LIN {X 89.539,Y 95.885,Z 82.299,A 180.000,B 0.000,C 180.000} C_DIS
LIN {X 89.506,Y 96.036,Z 82.293,A 180.000,B 0.000,C 180.000} C_DIS
LIN {X 89.491,Y 96.111,Z 82.291,A 180.000,B 0.000,C 180.000} C_DIS
LIN {X 89.478,Y 96.187,Z 82.288,A 180.000,B 0.000,C 180.000} C_DIS
LIN {X 89.454,Y 96.341,Z 82.283,A 180.000,B 0.000,C 180.000} C_DIS
LIN {X 89.442,Y 96.417,Z 82.280,A 180.000,B 0.000,C 180.000} C_DIS
LIN {X 89.431,Y 96.495,Z 82.277,A 180.000,B 0.000,C 180.000} C_DIS
LIN {X 89.420,Y 96.572,Z 82.274,A 180.000,B 0.000,C 180.000} C_DIS
LIN {X 89.409,Y 96.649,Z 82.272,A 180.000,B 0.000,C 180.000} C_DIS
LIN {X 89.400,Y 96.727,Z 82.269,A 180.000,B 0.000,C 180.000} C_DIS
LIN {X 89.392,Y 96.804,Z 82.266,A 180.000,B 0.000,C 180.000} C_DIS
LIN {X 89.376,Y 96.958,Z 82.261,A 180.000,B 0.000,C 180.000} C_DIS
LIN {X 89.369,Y 97.035,Z 82.258,A 180.000,B 0.000,C 180.000} C_DIS
LIN {X 89.365,Y 97.112,Z 82.255,A 180.000,B 0.000,C 180.000} C_DIS
LIN {X 89.358,Y 97.267,Z 82.250,A 180.000,B 0.000,C 180.000} C_DIS
LIN {X 89.355,Y 97.344,Z 82.247,A 180.000,B 0.000,C 180.000} C_DIS
LIN {X 89.353,Y 97.422,Z 82.245,A 180.000,B 0.000,C 180.000} C_DIS
LIN {X 89.351,Y 97.577,Z 82.239,A 180.000,B 0.000,C 180.000} C_DIS
LIN {X 89.350,Y 97.654,Z 82.236,A 180.000,B 0.000,C 180.000} C_DIS
LIN {X 89.351,Y 97.732,Z 82.234,A 180.000,B 0.000,C 180.000} C_DIS
LIN {X 89.353,Y 97.888,Z 82.228,A 180.000,B 0.000,C 180.000} C_DIS
LIN {X 89.354,Y 97.965,Z 82.226,A 180.000,B 0.000,C 180.000} C_DIS
LIN {X 89.359,Y 98.043,Z 82.223,A 180.000,B 0.000,C 180.000} C_DIS
LIN {X 89.369,Y 98.199,Z 82.217,A 180.000,B 0.000,C 180.000} C_DIS
LIN {X 89.375,Y 98.277,Z 82.215,A 180.000,B 0.000,C 180.000} C_DIS
LIN {X 89.382,Y 98.354,Z 82.212,A 180.000,B 0.000,C 180.000} C_DIS
LIN {X 89.390,Y 98.432,Z 82.209,A 180.000,B 0.000,C 180.000} C_DIS
LIN {X 89.398,Y 98.509,Z 82.207,A 180.000,B 0.000,C 180.000} C_DIS
LIN {X 89.407,Y 98.586,Z 82.204,A 180.000,B 0.000,C 180.000} C_DIS
LIN {X 89.416,Y 98.663,Z 82.201,A 180.000,B 0.000,C 180.000} C_DIS
LIN {X 89.436,Y 98.817,Z 82.196,A 180.000,B 0.000,C 180.000} C_DIS
LIN {X 89.446,Y 98.894,Z 82.193,A 180.000,B 0.000,C 180.000} C_DIS
LIN {X 89.459,Y 98.971,Z 82.190,A 180.000,B 0.000,C 180.000} C_DIS
LIN {X 89.487,Y 99.125,Z 82.185,A 180.000,B 0.000,C 180.000} C_DIS
LIN {X 89.501,Y 99.202,Z 82.182,A 180.000,B 0.000,C 180.000} C_DIS
LIN {X 89.516,Y 99.278,Z 82.180,A 180.000,B 0.000,C 180.000} C_DIS
LIN {X 89.534,Y 99.354,Z 82.177,A 180.000,B 0.000,C 180.000} C_DIS
LIN {X 89.552,Y 99.430,Z 82.174,A 180.000,B 0.000,C 180.000} C_DIS
LIN {X 89.570,Y 99.506,Z 82.172,A 180.000,B 0.000,C 180.000} C_DIS
LIN {X 89.589,Y 99.581,Z 82.169,A 180.000,B 0.000,C 180.000} C_DIS
LIN {X 89.607,Y 99.657,Z 82.167,A 180.000,B 0.000,C 180.000} C_DIS
LIN {X 89.625,Y 99.733,Z 82.164,A 180.000,B 0.000,C 180.000} C_DIS
LIN {X 89.644,Y 99.809,Z 82.161,A 180.000,B 0.000,C 180.000} C_DIS
LIN {X 89.665,Y 99.884,Z 82.159,A 180.000,B 0.000,C 180.000} C_DIS
LIN {X 89.688,Y 99.958,Z 82.156,A 180.000,B 0.000,C 180.000} C_DIS
LIN {X 89.733,Y 100.107,Z 82.151,A 180.000,B 0.000,C 180.000} C_DIS
LIN {X 89.783,Y 100.256,Z 82.146,A 180.000,B 0.000,C 180.000} C_DIS
LIN {X 89.837,Y 100.403,Z 82.141,A 180.000,B 0.000,C 180.000} C_DIS
LIN {X 89.892,Y 100.550,Z 82.137,A 180.000,B 0.000,C 180.000} C_DIS
LIN {X 89.947,Y 100.696,Z 82.132,A 180.000,B 0.000,C 180.000} C_DIS
LIN {X 90.008,Y 100.840,Z 82.127,A 180.000,B 0.000,C 180.000} C_DIS
LIN {X 90.070,Y 100.983,Z 82.123,A 180.000,B 0.000,C 180.000} C_DIS
LIN {X 90.136,Y 101.125,Z 82.118,A 180.000,B 0.000,C 180.000} C_DIS
LIN {X 90.206,Y 101.265,Z 82.113,A 180.000,B 0.000,C 180.000} C_DIS
LIN {X 90.277,Y 101.404,Z 82.109,A 180.000,B 0.000,C 180.000} C_DIS
LIN {X 90.351,Y 101.542,Z 82.105,A 180.000,B 0.000,C 180.000} C_DIS
LIN {X 90.428,Y 101.679,Z 82.100,A 180.000,B 0.000,C 180.000} C_DIS
LIN {X 90.506,Y 101.815,Z 82.096,A 180.000,B 0.000,C 180.000} C_DIS
LIN {X 90.587,Y 101.949,Z 82.092,A 180.000,B 0.000,C 180.000} C_DIS
LIN {X 90.673,Y 102.080,Z 82.088,A 180.000,B 0.000,C 180.000} C_DIS
LIN {X 90.760,Y 102.210,Z 82.084,A 180.000,B 0.000,C 180.000} C_DIS
LIN {X 90.851,Y 102.338,Z 82.080,A 180.000,B 0.000,C 180.000} C_DIS
LIN {X 90.943,Y 102.465,Z 82.076,A 180.000,B 0.000,C 180.000} C_DIS
LIN {X 91.036,Y 102.592,Z 82.072,A 180.000,B 0.000,C 180.000} C_DIS
LIN {X 91.132,Y 102.716,Z 82.069,A 180.000,B 0.000,C 180.000} C_DIS
LIN {X 91.232,Y 102.836,Z 82.065,A 180.000,B 0.000,C 180.000} C_DIS
LIN {X 91.333,Y 102.956,Z 82.062,A 180.000,B 0.000,C 180.000} C_DIS
LIN {X 91.439,Y 103.072,Z 82.058,A 180.000,B 0.000,C 180.000} C_DIS
LIN {X 91.546,Y 103.187,Z 82.055,A 180.000,B 0.000,C 180.000} C_DIS
LIN {X 91.653,Y 103.303,Z 82.052,A 180.000,B 0.000,C 180.000} C_DIS
LIN {X 91.762,Y 103.415,Z 82.048,A 180.000,B 0.000,C 180.000} C_DIS
LIN {X 91.875,Y 103.524,Z 82.045,A 180.000,B 0.000,C 180.000} C_DIS
LIN {X 91.990,Y 103.632,Z 82.042,A 180.000,B 0.000,C 180.000} C_DIS
LIN {X 92.108,Y 103.734,Z 82.040,A 180.000,B 0.000,C 180.000} C_DIS
LIN {X 92.228,Y 103.837,Z 82.037,A 180.000,B 0.000,C 180.000} C_DIS
LIN {X 92.348,Y 103.938,Z 82.034,A 180.000,B 0.000,C 180.000} C_DIS
LIN {X 92.470,Y 104.037,Z 82.031,A 180.000,B 0.000,C 180.000} C_DIS
LIN {X 92.595,Y 104.133,Z 82.029,A 180.000,B 0.000,C 180.000} C_DIS
LIN {X 92.851,Y 104.316,Z 82.024,A 180.000,B 0.000,C 180.000} C_DIS
LIN {X 93.113,Y 104.489,Z 82.020,A 180.000,B 0.000,C 180.000} C_DIS
LIN {X 93.381,Y 104.654,Z 82.016,A 180.000,B 0.000,C 180.000} C_DIS
LIN {X 93.656,Y 104.807,Z 82.012,A 180.000,B 0.000,C 180.000} C_DIS
LIN {X 93.937,Y 104.948,Z 82.009,A 180.000,B 0.000,C 180.000} C_DIS
LIN {X 94.223,Y 105.081,Z 82.006,A 180.000,B 0.000,C 180.000} C_DIS
LIN {X 94.514,Y 105.202,Z 82.004,A 180.000,B 0.000,C 180.000} C_DIS
LIN {X 94.809,Y 105.309,Z 82.002,A 180.000,B 0.000,C 180.000} C_DIS
LIN {X 95.109,Y 105.407,Z 82.001,A 180.000,B 0.000,C 180.000} C_DIS
LIN {X 95.412,Y 105.494,Z 82.000,A 180.000,B 0.000,C 180.000} C_DIS
LIN {X 95.718,Y 105.567,Z 82.000,A 180.000,B 0.000,C 180.000} C_DIS
LIN {X 95.782,Y 105.580,Z 82.000,A 180.000,B 0.000,C 180.000} C_DIS
; Cutting Move Starts
LIN {X 95.824,Y 105.588,Z 82.000,A 180.000,B 0.000,C 180.000} C_DIS
LIN {X 96.003,Y 105.623,Z 82.000,A 180.000,B 0.000,C 180.000} C_DIS
LIN {X 96.177,Y 105.656,Z 82.000,A 180.000,B 0.000,C 180.000} C_DIS
LIN {X 96.181,Y 105.657,Z 82.000,A 180.000,B 0.000,C 180.000} C_DIS
LIN {X 96.360,Y 105.683,Z 82.000,A 180.000,B 0.000,C 180.000} C_DIS
LIN {X 96.539,Y 105.708,Z 82.000,A 180.000,B 0.000,C 180.000} C_DIS
LIN {X 96.718,Y 105.724,Z 82.000,A 180.000,B 0.000,C 180.000} C_DIS
LIN {X 96.897,Y 105.739,Z 82.000,A 180.000,B 0.000,C 180.000} C_DIS
LIN {X 97.075,Y 105.750,Z 82.000,A 180.000,B 0.000,C 180.000} C_DIS
LIN {X 97.254,Y 105.758,Z 82.000,A 180.000,B 0.000,C 180.000} C_DIS
LIN {X 97.433,Y 105.763,Z 82.000,A 180.000,B 0.000,C 180.000} C_DIS
LIN {X 97.612,Y 105.762,Z 82.000,A 180.000,B 0.000,C 180.000} C_DIS
LIN {X 97.790,Y 105.757,Z 82.000,A 180.000,B 0.000,C 180.000} C_DIS
LIN {X 97.969,Y 105.748,Z 82.000,A 180.000,B 0.000,C 180.000} C_DIS
LIN {X 98.148,Y 105.736,Z 82.000,A 180.000,B 0.000,C 180.000} C_DIS
LIN {X 98.327,Y 105.721,Z 82.000,A 180.000,B 0.000,C 180.000} C_DIS
LIN {X 98.505,Y 105.702,Z 82.000,A 180.000,B 0.000,C 180.000} C_DIS
LIN {X 98.684,Y 105.677,Z 82.000,A 180.000,B 0.000,C 180.000} C_DIS
LIN {X 98.823,Y 105.656,Z 82.000,A 180.000,B 0.000,C 180.000} C_DIS
LIN {X 98.863,Y 105.649,Z 82.000,A 180.000,B 0.000,C 180.000} C_DIS
LIN {X 99.042,Y 105.615,Z 82.000,A 180.000,B 0.000,C 180.000} C_DIS
LIN {X 99.221,Y 105.580,Z 82.000,A 180.000,B 0.000,C 180.000} C_DIS
LIN {X 99.399,Y 105.542,Z 82.000,A 180.000,B 0.000,C 180.000} C_DIS
LIN {X 99.578,Y 105.497,Z 82.000,A 180.000,B 0.000,C 180.000} C_DIS
LIN {X 99.654,Y 105.477,Z 82.000,A 180.000,B 0.000,C 180.000} C_DIS
LIN {X 99.757,Y 105.449,Z 82.000,A 180.000,B 0.000,C 180.000} C_DIS
LIN {X 99.936,Y 105.393,Z 82.000,A 180.000,B 0.000,C 180.000} C_DIS
LIN {X 100.114,Y 105.335,Z 82.000,A 180.000,B 0.000,C 180.000} C_DIS
LIN {X 100.227,Y 105.299,Z 82.000,A 180.000,B 0.000,C 180.000} C_DIS
LIN {X 100.293,Y 105.277,Z 82.000,A 180.000,B 0.000,C 180.000} C_DIS
LIN {X 100.472,Y 105.209,Z 82.000,A 180.000,B 0.000,C 180.000} C_DIS
LIN {X 100.651,Y 105.140,Z 82.000,A 180.000,B 0.000,C 180.000} C_DIS
LIN {X 100.696,Y 105.120,Z 82.000,A 180.000,B 0.000,C 180.000} C_DIS
LIN {X 100.829,Y 105.060,Z 82.000,A 180.000,B 0.000,C 180.000} C_DIS
LIN {X 101.008,Y 104.979,Z 82.000,A 180.000,B 0.000,C 180.000} C_DIS
LIN {X 101.088,Y 104.941,Z 82.000,A 180.000,B 0.000,C 180.000} C_DIS
LIN {X 101.187,Y 104.894,Z 82.000,A 180.000,B 0.000,C 180.000} C_DIS
LIN {X 101.366,Y 104.802,Z 82.000,A 180.000,B 0.000,C 180.000} C_DIS
LIN {X 101.443,Y 104.762,Z 82.000,A 180.000,B 0.000,C 180.000} C_DIS
LIN {X 101.545,Y 104.706,Z 82.000,A 180.000,B 0.000,C 180.000} C_DIS
LIN {X 101.752,Y 104.584,Z 82.000,A 180.000,B 0.000,C 180.000} C_DIS
LIN {X 101.902,Y 104.490,Z 82.000,A 180.000,B 0.000,C 180.000} C_DIS
LIN {X 102.036,Y 104.405,Z 82.000,A 180.000,B 0.000,C 180.000} C_DIS
LIN {X 102.081,Y 104.375,Z 82.000,A 180.000,B 0.000,C 180.000} C_DIS
LIN {X 102.260,Y 104.255,Z 82.000,A 180.000,B 0.000,C 180.000} C_DIS
LIN {X 102.302,Y 104.226,Z 82.000,A 180.000,B 0.000,C 180.000} C_DIS
LIN {X 102.438,Y 104.124,Z 82.000,A 180.000,B 0.000,C 180.000} C_DIS
LIN {X 102.540,Y 104.047,Z 82.000,A 180.000,B 0.000,C 180.000} C_DIS
LIN {X 102.617,Y 103.987,Z 82.000,A 180.000,B 0.000,C 180.000} C_DIS
LIN {X 102.760,Y 103.869,Z 82.000,A 180.000,B 0.000,C 180.000} C_DIS
LIN {X 102.796,Y 103.839,Z 82.000,A 180.000,B 0.000,C 180.000} C_DIS
LIN {X 102.975,Y 103.688,Z 82.000,A 180.000,B 0.000,C 180.000} C_DIS
LIN {X 103.153,Y 103.526,Z 82.000,A 180.000,B 0.000,C 180.000} C_DIS
LIN {X 103.169,Y 103.511,Z 82.000,A 180.000,B 0.000,C 180.000} C_DIS
LIN {X 103.332,Y 103.353,Z 82.000,A 180.000,B 0.000,C 180.000} C_DIS
LIN {X 103.353,Y 103.332,Z 82.000,A 180.000,B 0.000,C 180.000} C_DIS
LIN {X 103.511,Y 103.165,Z 82.000,A 180.000,B 0.000,C 180.000} C_DIS
LIN {X 103.522,Y 103.153,Z 82.000,A 180.000,B 0.000,C 180.000} C_DIS
LIN {X 103.689,Y 102.975,Z 82.000,A 180.000,B 0.000,C 180.000} C_DIS
LIN {X 103.690,Y 102.974,Z 82.000,A 180.000,B 0.000,C 180.000} C_DIS
LIN {X 103.842,Y 102.796,Z 82.000,A 180.000,B 0.000,C 180.000} C_DIS
LIN {X 103.869,Y 102.765,Z 82.000,A 180.000,B 0.000,C 180.000} C_DIS
LIN {X 103.988,Y 102.617,Z 82.000,A 180.000,B 0.000,C 180.000} C_DIS
LIN {X 104.122,Y 102.438,Z 82.000,A 180.000,B 0.000,C 180.000} C_DIS
LIN {X 104.226,Y 102.296,Z 82.000,A 180.000,B 0.000,C 180.000} C_DIS
LIN {X 104.253,Y 102.260,Z 82.000,A 180.000,B 0.000,C 180.000} C_DIS
LIN {X 104.376,Y 102.081,Z 82.000,A 180.000,B 0.000,C 180.000} C_DIS
LIN {X 104.405,Y 102.037,Z 82.000,A 180.000,B 0.000,C 180.000} C_DIS
LIN {X 104.494,Y 101.902,Z 82.000,A 180.000,B 0.000,C 180.000} C_DIS
LIN {X 104.584,Y 101.752,Z 82.000,A 180.000,B 0.000,C 180.000} C_DIS
LIN {X 104.601,Y 101.723,Z 82.000,A 180.000,B 0.000,C 180.000} C_DIS
LIN {X 104.703,Y 101.545,Z 82.000,A 180.000,B 0.000,C 180.000} C_DIS
LIN {X 104.762,Y 101.437,Z 82.000,A 180.000,B 0.000,C 180.000} C_DIS
LIN {X 104.801,Y 101.366,Z 82.000,A 180.000,B 0.000,C 180.000} C_DIS
LIN {X 104.894,Y 101.187,Z 82.000,A 180.000,B 0.000,C 180.000} C_DIS
LIN {X 104.941,Y 101.095,Z 82.000,A 180.000,B 0.000,C 180.000} C_DIS
LIN {X 104.982,Y 101.008,Z 82.000,A 180.000,B 0.000,C 180.000} C_DIS
LIN {X 105.062,Y 100.829,Z 82.000,A 180.000,B 0.000,C 180.000} C_DIS
LIN {X 105.120,Y 100.693,Z 82.000,A 180.000,B 0.000,C 180.000} C_DIS
LIN {X 105.137,Y 100.651,Z 82.000,A 180.000,B 0.000,C 180.000} C_DIS
LIN {X 105.207,Y 100.472,Z 82.000,A 180.000,B 0.000,C 180.000} C_DIS
LIN {X 105.276,Y 100.293,Z 82.000,A 180.000,B 0.000,C 180.000} C_DIS
LIN {X 105.299,Y 100.232,Z 82.000,A 180.000,B 0.000,C 180.000} C_DIS
LIN {X 105.339,Y 100.114,Z 82.000,A 180.000,B 0.000,C 180.000} C_DIS
LIN {X 105.396,Y 99.936,Z 82.000,A 180.000,B 0.000,C 180.000} C_DIS
LIN {X 105.448,Y 99.757,Z 82.000,A 180.000,B 0.000,C 180.000} C_DIS
LIN {X 105.494,Y 99.578,Z 82.000,A 180.000,B 0.000,C 180.000} C_DIS
LIN {X 105.540,Y 99.399,Z 82.000,A 180.000,B 0.000,C 180.000} C_DIS
LIN {X 105.582,Y 99.221,Z 82.000,A 180.000,B 0.000,C 180.000} C_DIS
LIN {X 105.618,Y 99.042,Z 82.000,A 180.000,B 0.000,C 180.000} C_DIS
LIN {X 105.650,Y 98.863,Z 82.000,A 180.000,B 0.000,C 180.000} C_DIS
LIN {X 105.656,Y 98.819,Z 82.000,A 180.000,B 0.000,C 180.000} C_DIS
LIN {X 105.675,Y 98.684,Z 82.000,A 180.000,B 0.000,C 180.000} C_DIS
LIN {X 105.699,Y 98.505,Z 82.000,A 180.000,B 0.000,C 180.000} C_DIS
LIN {X 105.721,Y 98.327,Z 82.000,A 180.000,B 0.000,C 180.000} C_DIS
LIN {X 105.737,Y 98.148,Z 82.000,A 180.000,B 0.000,C 180.000} C_DIS
LIN {X 105.751,Y 97.969,Z 82.000,A 180.000,B 0.000,C 180.000} C_DIS
LIN {X 105.757,Y 97.790,Z 82.000,A 180.000,B 0.000,C 180.000} C_DIS
LIN {X 105.761,Y 97.612,Z 82.000,A 180.000,B 0.000,C 180.000} C_DIS
LIN {X 105.761,Y 97.433,Z 82.000,A 180.000,B 0.000,C 180.000} C_DIS
LIN {X 105.758,Y 97.254,Z 82.000,A 180.000,B 0.000,C 180.000} C_DIS
LIN {X 105.753,Y 97.075,Z 82.000,A 180.000,B 0.000,C 180.000} C_DIS
LIN {X 105.741,Y 96.897,Z 82.000,A 180.000,B 0.000,C 180.000} C_DIS
LIN {X 105.726,Y 96.718,Z 82.000,A 180.000,B 0.000,C 180.000} C_DIS
LIN {X 105.705,Y 96.539,Z 82.000,A 180.000,B 0.000,C 180.000} C_DIS
LIN {X 105.682,Y 96.360,Z 82.000,A 180.000,B 0.000,C 180.000} C_DIS
LIN {X 105.656,Y 96.181,Z 82.000,A 180.000,B 0.000,C 180.000} C_DIS
LIN {X 105.627,Y 96.003,Z 82.000,A 180.000,B 0.000,C 180.000} C_DIS
LIN {X 105.591,Y 95.824,Z 82.000,A 180.000,B 0.000,C 180.000} C_DIS
LIN {X 105.551,Y 95.645,Z 82.000,A 180.000,B 0.000,C 180.000} C_DIS
LIN {X 105.505,Y 95.466,Z 82.000,A 180.000,B 0.000,C 180.000} C_DIS
LIN {X 105.477,Y 95.359,Z 82.000,A 180.000,B 0.000,C 180.000} C_DIS
LIN {X 105.459,Y 95.288,Z 82.000,A 180.000,B 0.000,C 180.000} C_DIS
LIN {X 105.410,Y 95.109,Z 82.000,A 180.000,B 0.000,C 180.000} C_DIS
LIN {X 105.353,Y 94.930,Z 82.000,A 180.000,B 0.000,C 180.000} C_DIS
LIN {X 105.299,Y 94.768,Z 82.000,A 180.000,B 0.000,C 180.000} C_DIS
LIN {X 105.292,Y 94.751,Z 82.000,A 180.000,B 0.000,C 180.000} C_DIS
LIN {X 105.224,Y 94.573,Z 82.000,A 180.000,B 0.000,C 180.000} C_DIS
LIN {X 105.154,Y 94.394,Z 82.000,A 180.000,B 0.000,C 180.000} C_DIS
LIN {X 105.120,Y 94.307,Z 82.000,A 180.000,B 0.000,C 180.000} C_DIS
LIN {X 105.082,Y 94.215,Z 82.000,A 180.000,B 0.000,C 180.000} C_DIS
LIN {X 105.002,Y 94.036,Z 82.000,A 180.000,B 0.000,C 180.000} C_DIS
LIN {X 104.941,Y 93.905,Z 82.000,A 180.000,B 0.000,C 180.000} C_DIS
LIN {X 104.917,Y 93.857,Z 82.000,A 180.000,B 0.000,C 180.000} C_DIS
LIN {X 104.825,Y 93.679,Z 82.000,A 180.000,B 0.000,C 180.000} C_DIS
LIN {X 104.762,Y 93.563,Z 82.000,A 180.000,B 0.000,C 180.000} C_DIS
LIN {X 104.728,Y 93.500,Z 82.000,A 180.000,B 0.000,C 180.000} C_DIS
LIN {X 104.627,Y 93.321,Z 82.000,A 180.000,B 0.000,C 180.000} C_DIS
LIN {X 104.584,Y 93.248,Z 82.000,A 180.000,B 0.000,C 180.000} C_DIS
LIN {X 104.521,Y 93.142,Z 82.000,A 180.000,B 0.000,C 180.000} C_DIS
LIN {X 104.406,Y 92.964,Z 82.000,A 180.000,B 0.000,C 180.000} C_DIS
LIN {X 104.405,Y 92.963,Z 82.000,A 180.000,B 0.000,C 180.000} C_DIS
LIN {X 104.285,Y 92.785,Z 82.000,A 180.000,B 0.000,C 180.000} C_DIS
LIN {X 104.226,Y 92.704,Z 82.000,A 180.000,B 0.000,C 180.000} C_DIS
LIN {X 104.155,Y 92.606,Z 82.000,A 180.000,B 0.000,C 180.000} C_DIS
LIN {X 104.047,Y 92.462,Z 82.000,A 180.000,B 0.000,C 180.000} C_DIS
LIN {X 104.021,Y 92.427,Z 82.000,A 180.000,B 0.000,C 180.000} C_DIS
LIN {X 103.880,Y 92.249,Z 82.000,A 180.000,B 0.000,C 180.000} C_DIS
LIN {X 103.869,Y 92.235,Z 82.000,A 180.000,B 0.000,C 180.000} C_DIS
LIN {X 103.728,Y 92.070,Z 82.000,A 180.000,B 0.000,C 180.000} C_DIS
LIN {X 103.690,Y 92.026,Z 82.000,A 180.000,B 0.000,C 180.000} C_DIS
LIN {X 103.563,Y 91.891,Z 82.000,A 180.000,B 0.000,C 180.000} C_DIS
LIN {X 103.511,Y 91.835,Z 82.000,A 180.000,B 0.000,C 180.000} C_DIS
LIN {X 103.395,Y 91.712,Z 82.000,A 180.000,B 0.000,C 180.000} C_DIS
LIN {X 103.332,Y 91.647,Z 82.000,A 180.000,B 0.000,C 180.000} C_DIS
LIN {X 103.216,Y 91.533,Z 82.000,A 180.000,B 0.000,C 180.000} C_DIS
LIN {X 103.153,Y 91.474,Z 82.000,A 180.000,B 0.000,C 180.000} C_DIS
LIN {X 103.025,Y 91.355,Z 82.000,A 180.000,B 0.000,C 180.000} C_DIS
LIN {X 102.975,Y 91.312,Z 82.000,A 180.000,B 0.000,C 180.000} C_DIS
LIN {X 102.814,Y 91.176,Z 82.000,A 180.000,B 0.000,C 180.000} C_DIS
LIN {X 102.796,Y 91.161,Z 82.000,A 180.000,B 0.000,C 180.000} C_DIS
LIN {X 102.617,Y 91.013,Z 82.000,A 180.000,B 0.000,C 180.000} C_DIS
LIN {X 102.598,Y 90.997,Z 82.000,A 180.000,B 0.000,C 180.000} C_DIS
LIN {X 102.438,Y 90.876,Z 82.000,A 180.000,B 0.000,C 180.000} C_DIS
LIN {X 102.362,Y 90.818,Z 82.000,A 180.000,B 0.000,C 180.000} C_DIS
LIN {X 102.260,Y 90.745,Z 82.000,A 180.000,B 0.000,C 180.000} C_DIS
LIN {X 102.103,Y 90.640,Z 82.000,A 180.000,B 0.000,C 180.000} C_DIS
LIN {X 102.081,Y 90.625,Z 82.000,A 180.000,B 0.000,C 180.000} C_DIS
LIN {X 101.902,Y 90.510,Z 82.000,A 180.000,B 0.000,C 180.000} C_DIS
LIN {X 101.825,Y 90.461,Z 82.000,A 180.000,B 0.000,C 180.000} C_DIS
LIN {X 101.723,Y 90.399,Z 82.000,A 180.000,B 0.000,C 180.000} C_DIS
LIN {X 101.545,Y 90.294,Z 82.000,A 180.000,B 0.000,C 180.000} C_DIS
LIN {X 101.524,Y 90.282,Z 82.000,A 180.000,B 0.000,C 180.000} C_DIS
LIN {X 101.366,Y 90.198,Z 82.000,A 180.000,B 0.000,C 180.000} C_DIS
LIN {X 101.187,Y 90.106,Z 82.000,A 180.000,B 0.000,C 180.000} C_DIS
LIN {X 101.182,Y 90.103,Z 82.000,A 180.000,B 0.000,C 180.000} C_DIS
LIN {X 101.008,Y 90.021,Z 82.000,A 180.000,B 0.000,C 180.000} C_DIS
LIN {X 100.829,Y 89.940,Z 82.000,A 180.000,B 0.000,C 180.000} C_DIS
LIN {X 100.796,Y 89.925,Z 82.000,A 180.000,B 0.000,C 180.000} C_DIS
LIN {X 100.651,Y 89.860,Z 82.000,A 180.000,B 0.000,C 180.000} C_DIS
LIN {X 100.472,Y 89.791,Z 82.000,A 180.000,B 0.000,C 180.000} C_DIS
LIN {X 100.355,Y 89.746,Z 82.000,A 180.000,B 0.000,C 180.000} C_DIS
LIN {X 100.293,Y 89.723,Z 82.000,A 180.000,B 0.000,C 180.000} C_DIS
LIN {X 100.114,Y 89.665,Z 82.000,A 180.000,B 0.000,C 180.000} C_DIS
LIN {X 99.936,Y 89.607,Z 82.000,A 180.000,B 0.000,C 180.000} C_DIS
LIN {X 99.810,Y 89.567,Z 82.000,A 180.000,B 0.000,C 180.000} C_DIS
LIN {X 99.757,Y 89.551,Z 82.000,A 180.000,B 0.000,C 180.000} C_DIS
LIN {X 99.578,Y 89.503,Z 82.000,A 180.000,B 0.000,C 180.000} C_DIS
LIN {X 99.399,Y 89.458,Z 82.000,A 180.000,B 0.000,C 180.000} C_DIS
LIN {X 99.221,Y 89.420,Z 82.000,A 180.000,B 0.000,C 180.000} C_DIS
LIN {X 99.058,Y 89.388,Z 82.000,A 180.000,B 0.000,C 180.000} C_DIS
LIN {X 98.863,Y 89.351,Z 82.000,A 180.000,B 0.000,C 180.000} C_DIS
LIN {X 98.684,Y 89.323,Z 82.000,A 180.000,B 0.000,C 180.000} C_DIS
LIN {X 98.505,Y 89.298,Z 82.000,A 180.000,B 0.000,C 180.000} C_DIS
LIN {X 98.327,Y 89.279,Z 82.000,A 180.000,B 0.000,C 180.000} C_DIS
LIN {X 98.148,Y 89.264,Z 82.000,A 180.000,B 0.000,C 180.000} C_DIS
LIN {X 97.969,Y 89.252,Z 82.000,A 180.000,B 0.000,C 180.000} C_DIS
LIN {X 97.790,Y 89.243,Z 82.000,A 180.000,B 0.000,C 180.000} C_DIS
LIN {X 97.612,Y 89.238,Z 82.000,A 180.000,B 0.000,C 180.000} C_DIS
LIN {X 97.433,Y 89.237,Z 82.000,A 180.000,B 0.000,C 180.000} C_DIS
LIN {X 97.254,Y 89.242,Z 82.000,A 180.000,B 0.000,C 180.000} C_DIS
LIN {X 97.075,Y 89.250,Z 82.000,A 180.000,B 0.000,C 180.000} C_DIS
LIN {X 96.897,Y 89.261,Z 82.000,A 180.000,B 0.000,C 180.000} C_DIS
LIN {X 96.718,Y 89.276,Z 82.000,A 180.000,B 0.000,C 180.000} C_DIS
LIN {X 96.539,Y 89.292,Z 82.000,A 180.000,B 0.000,C 180.000} C_DIS
LIN {X 96.360,Y 89.317,Z 82.000,A 180.000,B 0.000,C 180.000} C_DIS
LIN {X 96.181,Y 89.343,Z 82.000,A 180.000,B 0.000,C 180.000} C_DIS
LIN {X 96.003,Y 89.377,Z 82.000,A 180.000,B 0.000,C 180.000} C_DIS
LIN {X 95.942,Y 89.388,Z 82.000,A 180.000,B 0.000,C 180.000} C_DIS
LIN {X 95.824,Y 89.412,Z 82.000,A 180.000,B 0.000,C 180.000} C_DIS
LIN {X 95.645,Y 89.447,Z 82.000,A 180.000,B 0.000,C 180.000} C_DIS
LIN {X 95.466,Y 89.492,Z 82.000,A 180.000,B 0.000,C 180.000} C_DIS
LIN {X 95.288,Y 89.538,Z 82.000,A 180.000,B 0.000,C 180.000} C_DIS
LIN {X 95.190,Y 89.567,Z 82.000,A 180.000,B 0.000,C 180.000} C_DIS
LIN {X 95.109,Y 89.593,Z 82.000,A 180.000,B 0.000,C 180.000} C_DIS
LIN {X 94.930,Y 89.650,Z 82.000,A 180.000,B 0.000,C 180.000} C_DIS
LIN {X 94.751,Y 89.708,Z 82.000,A 180.000,B 0.000,C 180.000} C_DIS
LIN {X 94.645,Y 89.746,Z 82.000,A 180.000,B 0.000,C 180.000} C_DIS
LIN {X 94.573,Y 89.774,Z 82.000,A 180.000,B 0.000,C 180.000} C_DIS
LIN {X 94.394,Y 89.842,Z 82.000,A 180.000,B 0.000,C 180.000} C_DIS
LIN {X 94.215,Y 89.920,Z 82.000,A 180.000,B 0.000,C 180.000} C_DIS
LIN {X 94.204,Y 89.925,Z 82.000,A 180.000,B 0.000,C 180.000} C_DIS
LIN {X 94.036,Y 90.000,Z 82.000,A 180.000,B 0.000,C 180.000} C_DIS
LIN {X 93.857,Y 90.085,Z 82.000,A 180.000,B 0.000,C 180.000} C_DIS
LIN {X 93.818,Y 90.103,Z 82.000,A 180.000,B 0.000,C 180.000} C_DIS
LIN {X 93.679,Y 90.175,Z 82.000,A 180.000,B 0.000,C 180.000} C_DIS
LIN {X 93.500,Y 90.268,Z 82.000,A 180.000,B 0.000,C 180.000} C_DIS
LIN {X 93.476,Y 90.282,Z 82.000,A 180.000,B 0.000,C 180.000} C_DIS
LIN {X 93.321,Y 90.373,Z 82.000,A 180.000,B 0.000,C 180.000} C_DIS
LIN {X 93.175,Y 90.461,Z 82.000,A 180.000,B 0.000,C 180.000} C_DIS
LIN {X 93.142,Y 90.482,Z 82.000,A 180.000,B 0.000,C 180.000} C_DIS
LIN {X 92.964,Y 90.595,Z 82.000,A 180.000,B 0.000,C 180.000} C_DIS
LIN {X 92.897,Y 90.640,Z 82.000,A 180.000,B 0.000,C 180.000} C_DIS
LIN {X 92.785,Y 90.715,Z 82.000,A 180.000,B 0.000,C 180.000} C_DIS
LIN {X 92.638,Y 90.818,Z 82.000,A 180.000,B 0.000,C 180.000} C_DIS
LIN {X 92.606,Y 90.842,Z 82.000,A 180.000,B 0.000,C 180.000} C_DIS
LIN {X 92.427,Y 90.977,Z 82.000,A 180.000,B 0.000,C 180.000} C_DIS
LIN {X 92.402,Y 90.997,Z 82.000,A 180.000,B 0.000,C 180.000} C_DIS
LIN {X 92.249,Y 91.124,Z 82.000,A 180.000,B 0.000,C 180.000} C_DIS
LIN {X 92.186,Y 91.176,Z 82.000,A 180.000,B 0.000,C 180.000} C_DIS
LIN {X 92.070,Y 91.274,Z 82.000,A 180.000,B 0.000,C 180.000} C_DIS
LIN {X 91.975,Y 91.355,Z 82.000,A 180.000,B 0.000,C 180.000} C_DIS
LIN {X 91.891,Y 91.432,Z 82.000,A 180.000,B 0.000,C 180.000} C_DIS
LIN {X 91.784,Y 91.533,Z 82.000,A 180.000,B 0.000,C 180.000} C_DIS
LIN {X 91.712,Y 91.602,Z 82.000,A 180.000,B 0.000,C 180.000} C_DIS
LIN {X 91.605,Y 91.712,Z 82.000,A 180.000,B 0.000,C 180.000} C_DIS
LIN {X 91.533,Y 91.788,Z 82.000,A 180.000,B 0.000,C 180.000} C_DIS
LIN {X 91.437,Y 91.891,Z 82.000,A 180.000,B 0.000,C 180.000} C_DIS
LIN {X 91.355,Y 91.978,Z 82.000,A 180.000,B 0.000,C 180.000} C_DIS
LIN {X 91.272,Y 92.070,Z 82.000,A 180.000,B 0.000,C 180.000} C_DIS
LIN {X 91.176,Y 92.183,Z 82.000,A 180.000,B 0.000,C 180.000} C_DIS
LIN {X 91.120,Y 92.249,Z 82.000,A 180.000,B 0.000,C 180.000} C_DIS
LIN {X 90.997,Y 92.403,Z 82.000,A 180.000,B 0.000,C 180.000} C_DIS
LIN {X 90.979,Y 92.427,Z 82.000,A 180.000,B 0.000,C 180.000} C_DIS
LIN {X 90.845,Y 92.606,Z 82.000,A 180.000,B 0.000,C 180.000} C_DIS
LIN {X 90.818,Y 92.643,Z 82.000,A 180.000,B 0.000,C 180.000} C_DIS
LIN {X 90.715,Y 92.785,Z 82.000,A 180.000,B 0.000,C 180.000} C_DIS
LIN {X 90.640,Y 92.896,Z 82.000,A 180.000,B 0.000,C 180.000} C_DIS
LIN {X 90.594,Y 92.964,Z 82.000,A 180.000,B 0.000,C 180.000} C_DIS
LIN {X 90.479,Y 93.142,Z 82.000,A 180.000,B 0.000,C 180.000} C_DIS
LIN {X 90.461,Y 93.172,Z 82.000,A 180.000,B 0.000,C 180.000} C_DIS
LIN {X 90.373,Y 93.321,Z 82.000,A 180.000,B 0.000,C 180.000} C_DIS
LIN {X 90.282,Y 93.482,Z 82.000,A 180.000,B 0.000,C 180.000} C_DIS
LIN {X 90.272,Y 93.500,Z 82.000,A 180.000,B 0.000,C 180.000} C_DIS
LIN {X 90.175,Y 93.679,Z 82.000,A 180.000,B 0.000,C 180.000} C_DIS
LIN {X 90.083,Y 93.857,Z 82.000,A 180.000,B 0.000,C 180.000} C_DIS
LIN {X 89.998,Y 94.036,Z 82.000,A 180.000,B 0.000,C 180.000} C_DIS
LIN {X 89.925,Y 94.201,Z 82.000,A 180.000,B 0.000,C 180.000} C_DIS
LIN {X 89.918,Y 94.215,Z 82.000,A 180.000,B 0.000,C 180.000} C_DIS
LIN {X 89.846,Y 94.394,Z 82.000,A 180.000,B 0.000,C 180.000} C_DIS
LIN {X 89.776,Y 94.573,Z 82.000,A 180.000,B 0.000,C 180.000} C_DIS
LIN {X 89.746,Y 94.651,Z 82.000,A 180.000,B 0.000,C 180.000} C_DIS
LIN {X 89.708,Y 94.751,Z 82.000,A 180.000,B 0.000,C 180.000} C_DIS
LIN {X 89.647,Y 94.930,Z 82.000,A 180.000,B 0.000,C 180.000} C_DIS
LIN {X 89.590,Y 95.109,Z 82.000,A 180.000,B 0.000,C 180.000} C_DIS
LIN {X 89.567,Y 95.188,Z 82.000,A 180.000,B 0.000,C 180.000} C_DIS
LIN {X 89.541,Y 95.288,Z 82.000,A 180.000,B 0.000,C 180.000} C_DIS
LIN {X 89.495,Y 95.466,Z 82.000,A 180.000,B 0.000,C 180.000} C_DIS
LIN {X 89.449,Y 95.645,Z 82.000,A 180.000,B 0.000,C 180.000} C_DIS
LIN {X 89.409,Y 95.824,Z 82.000,A 180.000,B 0.000,C 180.000} C_DIS
LIN {X 89.388,Y 95.929,Z 82.000,A 180.000,B 0.000,C 180.000} C_DIS
LIN {X 89.373,Y 96.003,Z 82.000,A 180.000,B 0.000,C 180.000} C_DIS
LIN {X 89.344,Y 96.181,Z 82.000,A 180.000,B 0.000,C 180.000} C_DIS
LIN {X 89.318,Y 96.360,Z 82.000,A 180.000,B 0.000,C 180.000} C_DIS
LIN {X 89.295,Y 96.539,Z 82.000,A 180.000,B 0.000,C 180.000} C_DIS
LIN {X 89.274,Y 96.718,Z 82.000,A 180.000,B 0.000,C 180.000} C_DIS
LIN {X 89.259,Y 96.897,Z 82.000,A 180.000,B 0.000,C 180.000} C_DIS
LIN {X 89.247,Y 97.075,Z 82.000,A 180.000,B 0.000,C 180.000} C_DIS
LIN {X 89.242,Y 97.254,Z 82.000,A 180.000,B 0.000,C 180.000} C_DIS
LIN {X 89.239,Y 97.433,Z 82.000,A 180.000,B 0.000,C 180.000} C_DIS
LIN {X 89.239,Y 97.612,Z 82.000,A 180.000,B 0.000,C 180.000} C_DIS
LIN {X 89.243,Y 97.790,Z 82.000,A 180.000,B 0.000,C 180.000} C_DIS
LIN {X 89.249,Y 97.969,Z 82.000,A 180.000,B 0.000,C 180.000} C_DIS
LIN {X 89.263,Y 98.148,Z 82.000,A 180.000,B 0.000,C 180.000} C_DIS
LIN {X 89.279,Y 98.327,Z 82.000,A 180.000,B 0.000,C 180.000} C_DIS
LIN {X 89.301,Y 98.505,Z 82.000,A 180.000,B 0.000,C 180.000} C_DIS
LIN {X 89.325,Y 98.684,Z 82.000,A 180.000,B 0.000,C 180.000} C_DIS
LIN {X 89.350,Y 98.863,Z 82.000,A 180.000,B 0.000,C 180.000} C_DIS
LIN {X 89.382,Y 99.042,Z 82.000,A 180.000,B 0.000,C 180.000} C_DIS
LIN {X 89.418,Y 99.221,Z 82.000,A 180.000,B 0.000,C 180.000} C_DIS
LIN {X 89.460,Y 99.399,Z 82.000,A 180.000,B 0.000,C 180.000} C_DIS
LIN {X 89.506,Y 99.578,Z 82.000,A 180.000,B 0.000,C 180.000} C_DIS
LIN {X 89.552,Y 99.757,Z 82.000,A 180.000,B 0.000,C 180.000} C_DIS
LIN {X 89.567,Y 99.812,Z 82.000,A 180.000,B 0.000,C 180.000} C_DIS
LIN {X 89.604,Y 99.936,Z 82.000,A 180.000,B 0.000,C 180.000} C_DIS
LIN {X 89.661,Y 100.114,Z 82.000,A 180.000,B 0.000,C 180.000} C_DIS
LIN {X 89.724,Y 100.293,Z 82.000,A 180.000,B 0.000,C 180.000} C_DIS
LIN {X 89.793,Y 100.472,Z 82.000,A 180.000,B 0.000,C 180.000} C_DIS
LIN {X 89.863,Y 100.651,Z 82.000,A 180.000,B 0.000,C 180.000} C_DIS
LIN {X 89.925,Y 100.799,Z 82.000,A 180.000,B 0.000,C 180.000} C_DIS
LIN {X 90.018,Y 101.008,Z 82.000,A 180.000,B 0.000,C 180.000} C_DIS
LIN {X 90.103,Y 101.182,Z 82.000,A 180.000,B 0.000,C 180.000} C_DIS
LIN {X 90.106,Y 101.187,Z 82.000,A 180.000,B 0.000,C 180.000} C_DIS
LIN {X 90.199,Y 101.366,Z 82.000,A 180.000,B 0.000,C 180.000} C_DIS
LIN {X 90.282,Y 101.518,Z 82.000,A 180.000,B 0.000,C 180.000} C_DIS
LIN {X 90.297,Y 101.545,Z 82.000,A 180.000,B 0.000,C 180.000} C_DIS
LIN {X 90.399,Y 101.723,Z 82.000,A 180.000,B 0.000,C 180.000} C_DIS
LIN {X 90.461,Y 101.828,Z 82.000,A 180.000,B 0.000,C 180.000} C_DIS
LIN {X 90.506,Y 101.902,Z 82.000,A 180.000,B 0.000,C 180.000} C_DIS
LIN {X 90.624,Y 102.081,Z 82.000,A 180.000,B 0.000,C 180.000} C_DIS
LIN {X 90.640,Y 102.104,Z 82.000,A 180.000,B 0.000,C 180.000} C_DIS
LIN {X 90.747,Y 102.260,Z 82.000,A 180.000,B 0.000,C 180.000} C_DIS
LIN {X 90.818,Y 102.357,Z 82.000,A 180.000,B 0.000,C 180.000} C_DIS
LIN {X 90.878,Y 102.438,Z 82.000,A 180.000,B 0.000,C 180.000} C_DIS
LIN {X 91.012,Y 102.617,Z 82.000,A 180.000,B 0.000,C 180.000} C_DIS
LIN {X 91.158,Y 102.796,Z 82.000,A 180.000,B 0.000,C 180.000} C_DIS
LIN {X 91.176,Y 102.817,Z 82.000,A 180.000,B 0.000,C 180.000} C_DIS
LIN {X 91.311,Y 102.975,Z 82.000,A 180.000,B 0.000,C 180.000} C_DIS
LIN {X 91.355,Y 103.022,Z 82.000,A 180.000,B 0.000,C 180.000} C_DIS
LIN {X 91.478,Y 103.153,Z 82.000,A 180.000,B 0.000,C 180.000} C_DIS
LIN {X 91.533,Y 103.212,Z 82.000,A 180.000,B 0.000,C 180.000} C_DIS
LIN {X 91.647,Y 103.332,Z 82.000,A 180.000,B 0.000,C 180.000} C_DIS
LIN {X 91.712,Y 103.398,Z 82.000,A 180.000,B 0.000,C 180.000} C_DIS
LIN {X 91.831,Y 103.511,Z 82.000,A 180.000,B 0.000,C 180.000} C_DIS
LIN {X 91.891,Y 103.568,Z 82.000,A 180.000,B 0.000,C 180.000} C_DIS
LIN {X 92.027,Y 103.690,Z 82.000,A 180.000,B 0.000,C 180.000} C_DIS
LIN {X 92.070,Y 103.726,Z 82.000,A 180.000,B 0.000,C 180.000} C_DIS
LIN {X 92.240,Y 103.869,Z 82.000,A 180.000,B 0.000,C 180.000} C_DIS
LIN {X 92.249,Y 103.876,Z 82.000,A 180.000,B 0.000,C 180.000} C_DIS
LIN {X 92.427,Y 104.023,Z 82.000,A 180.000,B 0.000,C 180.000} C_DIS
LIN {X 92.460,Y 104.047,Z 82.000,A 180.000,B 0.000,C 180.000} C_DIS
LIN {X 92.606,Y 104.158,Z 82.000,A 180.000,B 0.000,C 180.000} C_DIS
LIN {X 92.698,Y 104.226,Z 82.000,A 180.000,B 0.000,C 180.000} C_DIS
LIN {X 92.785,Y 104.285,Z 82.000,A 180.000,B 0.000,C 180.000} C_DIS
LIN {X 92.964,Y 104.405,Z 82.000,A 180.000,B 0.000,C 180.000} C_DIS
LIN {X 93.142,Y 104.518,Z 82.000,A 180.000,B 0.000,C 180.000} C_DIS
LIN {X 93.248,Y 104.584,Z 82.000,A 180.000,B 0.000,C 180.000} C_DIS
LIN {X 93.321,Y 104.627,Z 82.000,A 180.000,B 0.000,C 180.000} C_DIS
LIN {X 93.500,Y 104.732,Z 82.000,A 180.000,B 0.000,C 180.000} C_DIS
LIN {X 93.557,Y 104.762,Z 82.000,A 180.000,B 0.000,C 180.000} C_DIS
LIN {X 93.679,Y 104.825,Z 82.000,A 180.000,B 0.000,C 180.000} C_DIS
LIN {X 93.857,Y 104.915,Z 82.000,A 180.000,B 0.000,C 180.000} C_DIS
LIN {X 94.036,Y 105.000,Z 82.000,A 180.000,B 0.000,C 180.000} C_DIS
LIN {X 94.215,Y 105.080,Z 82.000,A 180.000,B 0.000,C 180.000} C_DIS
LIN {X 94.304,Y 105.120,Z 82.000,A 180.000,B 0.000,C 180.000} C_DIS
LIN {X 94.394,Y 105.158,Z 82.000,A 180.000,B 0.000,C 180.000} C_DIS
LIN {X 94.573,Y 105.226,Z 82.000,A 180.000,B 0.000,C 180.000} C_DIS
LIN {X 94.751,Y 105.292,Z 82.000,A 180.000,B 0.000,C 180.000} C_DIS
LIN {X 94.773,Y 105.299,Z 82.000,A 180.000,B 0.000,C 180.000} C_DIS
LIN {X 94.930,Y 105.350,Z 82.000,A 180.000,B 0.000,C 180.000} C_DIS
LIN {X 95.109,Y 105.407,Z 82.000,A 180.000,B 0.000,C 180.000} C_DIS
LIN {X 95.288,Y 105.462,Z 82.000,A 180.000,B 0.000,C 180.000} C_DIS
LIN {X 95.346,Y 105.477,Z 82.000,A 180.000,B 0.000,C 180.000} C_DIS
LIN {X 95.466,Y 105.508,Z 82.000,A 180.000,B 0.000,C 180.000} C_DIS
LIN {X 95.645,Y 105.553,Z 82.000,A 180.000,B 0.000,C 180.000} C_DIS
LIN {X 95.782,Y 105.580,Z 82.000,A 180.000,B 0.000,C 180.000} C_DIS
; Link Move Starts
LIN {X 96.086,Y 105.639,Z 82.000,A 180.000,B 0.000,C 180.000} C_DIS
LIN {X 96.376,Y 105.686,Z 81.999,A 180.000,B 0.000,C 180.000} C_DIS
LIN {X 96.664,Y 105.721,Z 81.998,A 180.000,B 0.000,C 180.000} C_DIS
LIN {X 96.967,Y 105.745,Z 81.996,A 180.000,B 0.000,C 180.000} C_DIS
LIN {X 97.269,Y 105.761,Z 81.995,A 180.000,B 0.000,C 180.000} C_DIS
LIN {X 97.564,Y 105.767,Z 81.992,A 180.000,B 0.000,C 180.000} C_DIS
LIN {X 97.861,Y 105.759,Z 81.989,A 180.000,B 0.000,C 180.000} C_DIS
LIN {X 98.158,Y 105.741,Z 81.986,A 180.000,B 0.000,C 180.000} C_DIS
LIN {X 98.454,Y 105.717,Z 81.983,A 180.000,B 0.000,C 180.000} C_DIS
LIN {X 98.758,Y 105.677,Z 81.979,A 180.000,B 0.000,C 180.000} C_DIS
LIN {X 99.046,Y 105.626,Z 81.975,A 180.000,B 0.000,C 180.000} C_DIS
LIN {X 99.338,Y 105.570,Z 81.970,A 180.000,B 0.000,C 180.000} C_DIS
LIN {X 99.486,Y 105.536,Z 81.968,A 180.000,B 0.000,C 180.000} C_DIS
LIN {X 99.635,Y 105.499,Z 81.965,A 180.000,B 0.000,C 180.000} C_DIS
LIN {X 99.775,Y 105.462,Z 81.962,A 180.000,B 0.000,C 180.000} C_DIS
LIN {X 99.913,Y 105.420,Z 81.960,A 180.000,B 0.000,C 180.000} C_DIS
LIN {X 100.061,Y 105.374,Z 81.957,A 180.000,B 0.000,C 180.000} C_DIS
LIN {X 100.208,Y 105.328,Z 81.954,A 180.000,B 0.000,C 180.000} C_DIS
LIN {X 100.349,Y 105.281,Z 81.951,A 180.000,B 0.000,C 180.000} C_DIS
LIN {X 100.488,Y 105.229,Z 81.948,A 180.000,B 0.000,C 180.000} C_DIS
LIN {X 100.624,Y 105.178,Z 81.945,A 180.000,B 0.000,C 180.000} C_DIS
LIN {X 100.759,Y 105.122,Z 81.942,A 180.000,B 0.000,C 180.000} C_DIS
LIN {X 100.899,Y 105.061,Z 81.938,A 180.000,B 0.000,C 180.000} C_DIS
LIN {X 101.038,Y 104.998,Z 81.935,A 180.000,B 0.000,C 180.000} C_DIS
LIN {X 101.174,Y 104.936,Z 81.931,A 180.000,B 0.000,C 180.000} C_DIS
LIN {X 101.308,Y 104.870,Z 81.928,A 180.000,B 0.000,C 180.000} C_DIS
LIN {X 101.438,Y 104.805,Z 81.924,A 180.000,B 0.000,C 180.000} C_DIS
LIN {X 101.566,Y 104.736,Z 81.921,A 180.000,B 0.000,C 180.000} C_DIS
LIN {X 101.702,Y 104.658,Z 81.917,A 180.000,B 0.000,C 180.000} C_DIS
LIN {X 101.837,Y 104.580,Z 81.913,A 180.000,B 0.000,C 180.000} C_DIS
LIN {X 101.962,Y 104.502,Z 81.909,A 180.000,B 0.000,C 180.000} C_DIS
LIN {X 102.087,Y 104.424,Z 81.905,A 180.000,B 0.000,C 180.000} C_DIS
LIN {X 102.216,Y 104.340,Z 81.901,A 180.000,B 0.000,C 180.000} C_DIS
LIN {X 102.345,Y 104.255,Z 81.897,A 180.000,B 0.000,C 180.000} C_DIS
LIN {X 102.465,Y 104.167,Z 81.892,A 180.000,B 0.000,C 180.000} C_DIS
LIN {X 102.584,Y 104.079,Z 81.888,A 180.000,B 0.000,C 180.000} C_DIS
LIN {X 102.700,Y 103.989,Z 81.884,A 180.000,B 0.000,C 180.000} C_DIS
LIN {X 102.814,Y 103.897,Z 81.880,A 180.000,B 0.000,C 180.000} C_DIS
LIN {X 102.934,Y 103.799,Z 81.875,A 180.000,B 0.000,C 180.000} C_DIS
LIN {X 103.054,Y 103.700,Z 81.870,A 180.000,B 0.000,C 180.000} C_DIS
LIN {X 103.163,Y 103.603,Z 81.866,A 180.000,B 0.000,C 180.000} C_DIS
LIN {X 103.270,Y 103.504,Z 81.861,A 180.000,B 0.000,C 180.000} C_DIS
LIN {X 103.378,Y 103.402,Z 81.857,A 180.000,B 0.000,C 180.000} C_DIS
LIN {X 103.481,Y 103.296,Z 81.852,A 180.000,B 0.000,C 180.000} C_DIS
LIN {X 103.536,Y 103.240,Z 81.850,A 180.000,B 0.000,C 180.000} C_DIS
LIN {X 103.591,Y 103.184,Z 81.847,A 180.000,B 0.000,C 180.000} C_DIS
LIN {X 103.645,Y 103.128,Z 81.844,A 180.000,B 0.000,C 180.000} C_DIS
LIN {X 103.700,Y 103.071,Z 81.842,A 180.000,B 0.000,C 180.000} C_DIS
LIN {X 103.800,Y 102.963,Z 81.837,A 180.000,B 0.000,C 180.000} C_DIS
LIN {X 103.897,Y 102.852,Z 81.832,A 180.000,B 0.000,C 180.000} C_DIS
LIN {X 103.994,Y 102.740,Z 81.827,A 180.000,B 0.000,C 180.000} C_DIS
LIN {X 104.041,Y 102.683,Z 81.825,A 180.000,B 0.000,C 180.000} C_DIS
LIN {X 104.086,Y 102.624,Z 81.822,A 180.000,B 0.000,C 180.000} C_DIS
LIN {X 104.180,Y 102.504,Z 81.817,A 180.000,B 0.000,C 180.000} C_DIS
LIN {X 104.226,Y 102.443,Z 81.814,A 180.000,B 0.000,C 180.000} C_DIS
LIN {X 104.317,Y 102.322,Z 81.809,A 180.000,B 0.000,C 180.000} C_DIS
LIN {X 104.362,Y 102.262,Z 81.806,A 180.000,B 0.000,C 180.000} C_DIS
LIN {X 104.406,Y 102.201,Z 81.804,A 180.000,B 0.000,C 180.000} C_DIS
LIN {X 104.449,Y 102.139,Z 81.801,A 180.000,B 0.000,C 180.000} C_DIS
LIN {X 104.534,Y 102.015,Z 81.796,A 180.000,B 0.000,C 180.000} C_DIS
LIN {X 104.576,Y 101.952,Z 81.793,A 180.000,B 0.000,C 180.000} C_DIS
LIN {X 104.617,Y 101.888,Z 81.791,A 180.000,B 0.000,C 180.000} C_DIS
LIN {X 104.695,Y 101.760,Z 81.785,A 180.000,B 0.000,C 180.000} C_DIS
LIN {X 104.735,Y 101.695,Z 81.783,A 180.000,B 0.000,C 180.000} C_DIS
LIN {X 104.773,Y 101.630,Z 81.780,A 180.000,B 0.000,C 180.000} C_DIS
LIN {X 104.848,Y 101.500,Z 81.775,A 180.000,B 0.000,C 180.000} C_DIS
LIN {X 104.885,Y 101.435,Z 81.772,A 180.000,B 0.000,C 180.000} C_DIS
LIN {X 104.921,Y 101.369,Z 81.769,A 180.000,B 0.000,C 180.000} C_DIS
LIN {X 104.993,Y 101.234,Z 81.764,A 180.000,B 0.000,C 180.000} C_DIS
LIN {X 105.029,Y 101.167,Z 81.761,A 180.000,B 0.000,C 180.000} C_DIS
LIN {X 105.064,Y 101.099,Z 81.759,A 180.000,B 0.000,C 180.000} C_DIS
LIN {X 105.096,Y 101.032,Z 81.756,A 180.000,B 0.000,C 180.000} C_DIS
LIN {X 105.159,Y 100.897,Z 81.751,A 180.000,B 0.000,C 180.000} C_DIS
LIN {X 105.190,Y 100.830,Z 81.748,A 180.000,B 0.000,C 180.000} C_DIS
LIN {X 105.221,Y 100.760,Z 81.746,A 180.000,B 0.000,C 180.000} C_DIS
LIN {X 105.251,Y 100.689,Z 81.743,A 180.000,B 0.000,C 180.000} C_DIS
LIN {X 105.309,Y 100.547,Z 81.738,A 180.000,B 0.000,C 180.000} C_DIS
LIN {X 105.338,Y 100.476,Z 81.735,A 180.000,B 0.000,C 180.000} C_DIS
LIN {X 105.395,Y 100.334,Z 81.730,A 180.000,B 0.000,C 180.000} C_DIS
LIN {X 105.423,Y 100.264,Z 81.727,A 180.000,B 0.000,C 180.000} C_DIS
LIN {X 105.448,Y 100.194,Z 81.724,A 180.000,B 0.000,C 180.000} C_DIS
LIN {X 105.472,Y 100.123,Z 81.722,A 180.000,B 0.000,C 180.000} C_DIS
LIN {X 105.520,Y 99.982,Z 81.717,A 180.000,B 0.000,C 180.000} C_DIS
LIN {X 105.543,Y 99.910,Z 81.714,A 180.000,B 0.000,C 180.000} C_DIS
LIN {X 105.565,Y 99.838,Z 81.711,A 180.000,B 0.000,C 180.000} C_DIS
LIN {X 105.585,Y 99.766,Z 81.709,A 180.000,B 0.000,C 180.000} C_DIS
LIN {X 105.605,Y 99.693,Z 81.706,A 180.000,B 0.000,C 180.000} C_DIS
LIN {X 105.626,Y 99.618,Z 81.703,A 180.000,B 0.000,C 180.000} C_DIS
LIN {X 105.647,Y 99.542,Z 81.701,A 180.000,B 0.000,C 180.000} C_DIS
LIN {X 105.689,Y 99.391,Z 81.695,A 180.000,B 0.000,C 180.000} C_DIS
LIN {X 105.708,Y 99.319,Z 81.693,A 180.000,B 0.000,C 180.000} C_DIS
LIN {X 105.724,Y 99.246,Z 81.690,A 180.000,B 0.000,C 180.000} C_DIS
LIN {X 105.771,Y 99.028,Z 81.682,A 180.000,B 0.000,C 180.000} C_DIS
LIN {X 105.786,Y 98.955,Z 81.680,A 180.000,B 0.000,C 180.000} C_DIS
LIN {X 105.799,Y 98.882,Z 81.677,A 180.000,B 0.000,C 180.000} C_DIS
LIN {X 105.811,Y 98.809,Z 81.674,A 180.000,B 0.000,C 180.000} C_DIS
LIN {X 105.835,Y 98.655,Z 81.669,A 180.000,B 0.000,C 180.000} C_DIS
LIN {X 105.847,Y 98.578,Z 81.666,A 180.000,B 0.000,C 180.000} C_DIS
LIN {X 105.858,Y 98.501,Z 81.664,A 180.000,B 0.000,C 180.000} C_DIS
LIN {X 105.869,Y 98.426,Z 81.661,A 180.000,B 0.000,C 180.000} C_DIS
LIN {X 105.879,Y 98.352,Z 81.658,A 180.000,B 0.000,C 180.000} C_DIS
LIN {X 105.887,Y 98.277,Z 81.656,A 180.000,B 0.000,C 180.000} C_DIS
LIN {X 105.902,Y 98.127,Z 81.650,A 180.000,B 0.000,C 180.000} C_DIS
LIN {X 105.910,Y 98.053,Z 81.648,A 180.000,B 0.000,C 180.000} C_DIS
LIN {X 105.916,Y 97.979,Z 81.645,A 180.000,B 0.000,C 180.000} C_DIS
LIN {X 105.920,Y 97.904,Z 81.643,A 180.000,B 0.000,C 180.000} C_DIS
LIN {X 105.930,Y 97.675,Z 81.635,A 180.000,B 0.000,C 180.000} C_DIS
LIN {X 105.933,Y 97.598,Z 81.632,A 180.000,B 0.000,C 180.000} C_DIS
LIN {X 105.935,Y 97.443,Z 81.626,A 180.000,B 0.000,C 180.000} C_DIS
LIN {X 105.936,Y 97.366,Z 81.624,A 180.000,B 0.000,C 180.000} C_DIS
LIN {X 105.936,Y 97.288,Z 81.621,A 180.000,B 0.000,C 180.000} C_DIS
LIN {X 105.934,Y 97.137,Z 81.616,A 180.000,B 0.000,C 180.000} C_DIS
LIN {X 105.933,Y 97.061,Z 81.613,A 180.000,B 0.000,C 180.000} C_DIS
LIN {X 105.930,Y 96.986,Z 81.610,A 180.000,B 0.000,C 180.000} C_DIS
LIN {X 105.925,Y 96.910,Z 81.608,A 180.000,B 0.000,C 180.000} C_DIS
LIN {X 105.915,Y 96.759,Z 81.603,A 180.000,B 0.000,C 180.000} C_DIS
LIN {X 105.910,Y 96.683,Z 81.600,A 180.000,B 0.000,C 180.000} C_DIS
LIN {X 105.903,Y 96.607,Z 81.597,A 180.000,B 0.000,C 180.000} C_DIS
LIN {X 105.886,Y 96.456,Z 81.592,A 180.000,B 0.000,C 180.000} C_DIS
LIN {X 105.878,Y 96.380,Z 81.589,A 180.000,B 0.000,C 180.000} C_DIS
LIN {X 105.868,Y 96.302,Z 81.587,A 180.000,B 0.000,C 180.000} C_DIS
LIN {X 105.849,Y 96.147,Z 81.581,A 180.000,B 0.000,C 180.000} C_DIS
LIN {X 105.839,Y 96.069,Z 81.578,A 180.000,B 0.000,C 180.000} C_DIS
LIN {X 105.827,Y 95.995,Z 81.576,A 180.000,B 0.000,C 180.000} C_DIS
LIN {X 105.813,Y 95.921,Z 81.573,A 180.000,B 0.000,C 180.000} C_DIS
LIN {X 105.786,Y 95.773,Z 81.568,A 180.000,B 0.000,C 180.000} C_DIS
LIN {X 105.772,Y 95.699,Z 81.565,A 180.000,B 0.000,C 180.000} C_DIS
LIN {X 105.756,Y 95.625,Z 81.563,A 180.000,B 0.000,C 180.000} C_DIS
LIN {X 105.739,Y 95.552,Z 81.560,A 180.000,B 0.000,C 180.000} C_DIS
LIN {X 105.703,Y 95.403,Z 81.555,A 180.000,B 0.000,C 180.000} C_DIS
LIN {X 105.649,Y 95.177,Z 81.546,A 180.000,B 0.000,C 180.000} C_DIS
LIN {X 105.630,Y 95.103,Z 81.544,A 180.000,B 0.000,C 180.000} C_DIS
LIN {X 105.609,Y 95.030,Z 81.541,A 180.000,B 0.000,C 180.000} C_DIS
LIN {X 105.544,Y 94.811,Z 81.533,A 180.000,B 0.000,C 180.000} C_DIS
LIN {X 105.521,Y 94.740,Z 81.531,A 180.000,B 0.000,C 180.000} C_DIS
LIN {X 105.496,Y 94.668,Z 81.528,A 180.000,B 0.000,C 180.000} C_DIS
LIN {X 105.417,Y 94.451,Z 81.520,A 180.000,B 0.000,C 180.000} C_DIS
LIN {X 105.390,Y 94.378,Z 81.517,A 180.000,B 0.000,C 180.000} C_DIS
LIN {X 105.336,Y 94.233,Z 81.512,A 180.000,B 0.000,C 180.000} C_DIS
LIN {X 105.308,Y 94.162,Z 81.509,A 180.000,B 0.000,C 180.000} C_DIS
LIN {X 105.279,Y 94.092,Z 81.506,A 180.000,B 0.000,C 180.000} C_DIS
LIN {X 105.189,Y 93.883,Z 81.498,A 180.000,B 0.000,C 180.000} C_DIS
LIN {X 105.159,Y 93.815,Z 81.496,A 180.000,B 0.000,C 180.000} C_DIS
LIN {X 105.126,Y 93.747,Z 81.493,A 180.000,B 0.000,C 180.000} C_DIS
LIN {X 105.021,Y 93.537,Z 81.485,A 180.000,B 0.000,C 180.000} C_DIS
LIN {X 104.986,Y 93.467,Z 81.482,A 180.000,B 0.000,C 180.000} C_DIS
LIN {X 104.914,Y 93.333,Z 81.477,A 180.000,B 0.000,C 180.000} C_DIS
LIN {X 104.878,Y 93.265,Z 81.474,A 180.000,B 0.000,C 180.000} C_DIS
LIN {X 104.841,Y 93.199,Z 81.472,A 180.000,B 0.000,C 180.000} C_DIS
LIN {X 104.764,Y 93.064,Z 81.466,A 180.000,B 0.000,C 180.000} C_DIS
LIN {X 104.726,Y 92.997,Z 81.464,A 180.000,B 0.000,C 180.000} C_DIS
LIN {X 104.686,Y 92.931,Z 81.461,A 180.000,B 0.000,C 180.000} C_DIS
LIN {X 104.645,Y 92.867,Z 81.458,A 180.000,B 0.000,C 180.000} C_DIS
LIN {X 104.562,Y 92.739,Z 81.453,A 180.000,B 0.000,C 180.000} C_DIS
LIN {X 104.521,Y 92.676,Z 81.450,A 180.000,B 0.000,C 180.000} C_DIS
LIN {X 104.478,Y 92.612,Z 81.447,A 180.000,B 0.000,C 180.000} C_DIS
LIN {X 104.389,Y 92.485,Z 81.442,A 180.000,B 0.000,C 180.000} C_DIS
LIN {X 104.344,Y 92.421,Z 81.439,A 180.000,B 0.000,C 180.000} C_DIS
LIN {X 104.254,Y 92.298,Z 81.434,A 180.000,B 0.000,C 180.000} C_DIS
LIN {X 104.209,Y 92.236,Z 81.431,A 180.000,B 0.000,C 180.000} C_DIS
LIN {X 104.164,Y 92.175,Z 81.429,A 180.000,B 0.000,C 180.000} C_DIS
LIN {X 104.116,Y 92.114,Z 81.426,A 180.000,B 0.000,C 180.000} C_DIS
LIN {X 104.067,Y 92.054,Z 81.423,A 180.000,B 0.000,C 180.000} C_DIS
LIN {X 103.968,Y 91.933,Z 81.418,A 180.000,B 0.000,C 180.000} C_DIS
LIN {X 103.920,Y 91.874,Z 81.415,A 180.000,B 0.000,C 180.000} C_DIS
LIN {X 103.869,Y 91.817,Z 81.413,A 180.000,B 0.000,C 180.000} C_DIS
LIN {X 103.766,Y 91.703,Z 81.407,A 180.000,B 0.000,C 180.000} C_DIS
LIN {X 103.714,Y 91.646,Z 81.404,A 180.000,B 0.000,C 180.000} C_DIS
LIN {X 103.557,Y 91.475,Z 81.396,A 180.000,B 0.000,C 180.000} C_DIS
LIN {X 103.505,Y 91.419,Z 81.394,A 180.000,B 0.000,C 180.000} C_DIS
LIN {X 103.450,Y 91.364,Z 81.391,A 180.000,B 0.000,C 180.000} C_DIS
LIN {X 103.285,Y 91.203,Z 81.383,A 180.000,B 0.000,C 180.000} C_DIS
LIN {X 103.230,Y 91.150,Z 81.380,A 180.000,B 0.000,C 180.000} C_DIS
LIN {X 103.173,Y 91.099,Z 81.378,A 180.000,B 0.000,C 180.000} C_DIS
LIN {X 103.056,Y 90.997,Z 81.372,A 180.000,B 0.000,C 180.000} C_DIS
LIN {X 102.997,Y 90.946,Z 81.369,A 180.000,B 0.000,C 180.000} C_DIS
LIN {X 102.937,Y 90.895,Z 81.367,A 180.000,B 0.000,C 180.000} C_DIS
LIN {X 102.820,Y 90.794,Z 81.361,A 180.000,B 0.000,C 180.000} C_DIS
LIN {X 102.761,Y 90.745,Z 81.359,A 180.000,B 0.000,C 180.000} C_DIS
LIN {X 102.700,Y 90.697,Z 81.356,A 180.000,B 0.000,C 180.000} C_DIS
LIN {X 102.579,Y 90.603,Z 81.351,A 180.000,B 0.000,C 180.000} C_DIS
LIN {X 102.518,Y 90.555,Z 81.348,A 180.000,B 0.000,C 180.000} C_DIS
LIN {X 102.456,Y 90.509,Z 81.345,A 180.000,B 0.000,C 180.000} C_DIS
LIN {X 102.393,Y 90.465,Z 81.342,A 180.000,B 0.000,C 180.000} C_DIS
LIN {X 102.266,Y 90.377,Z 81.337,A 180.000,B 0.000,C 180.000} C_DIS
LIN {X 102.202,Y 90.333,Z 81.334,A 180.000,B 0.000,C 180.000} C_DIS
LIN {X 102.138,Y 90.290,Z 81.332,A 180.000,B 0.000,C 180.000} C_DIS
LIN {X 102.008,Y 90.205,Z 81.326,A 180.000,B 0.000,C 180.000} C_DIS
LIN {X 101.943,Y 90.163,Z 81.324,A 180.000,B 0.000,C 180.000} C_DIS
LIN {X 101.876,Y 90.122,Z 81.321,A 180.000,B 0.000,C 180.000} C_DIS
LIN {X 101.746,Y 90.042,Z 81.315,A 180.000,B 0.000,C 180.000} C_DIS
LIN {X 101.680,Y 90.002,Z 81.313,A 180.000,B 0.000,C 180.000} C_DIS
LIN {X 101.614,Y 89.964,Z 81.310,A 180.000,B 0.000,C 180.000} C_DIS
LIN {X 101.545,Y 89.927,Z 81.307,A 180.000,B 0.000,C 180.000} C_DIS
LIN {X 101.407,Y 89.853,Z 81.302,A 180.000,B 0.000,C 180.000} C_DIS
LIN {X 101.338,Y 89.816,Z 81.299,A 180.000,B 0.000,C 180.000} C_DIS
LIN {X 101.269,Y 89.781,Z 81.296,A 180.000,B 0.000,C 180.000} C_DIS
LIN {X 101.130,Y 89.713,Z 81.291,A 180.000,B 0.000,C 180.000} C_DIS
LIN {X 101.061,Y 89.680,Z 81.288,A 180.000,B 0.000,C 180.000} C_DIS
LIN {X 100.920,Y 89.614,Z 81.283,A 180.000,B 0.000,C 180.000} C_DIS
LIN {X 100.849,Y 89.581,Z 81.280,A 180.000,B 0.000,C 180.000} C_DIS
LIN {X 100.778,Y 89.549,Z 81.278,A 180.000,B 0.000,C 180.000} C_DIS
LIN {X 100.707,Y 89.518,Z 81.275,A 180.000,B 0.000,C 180.000} C_DIS
LIN {X 100.562,Y 89.461,Z 81.269,A 180.000,B 0.000,C 180.000} C_DIS
LIN {X 100.490,Y 89.432,Z 81.267,A 180.000,B 0.000,C 180.000} C_DIS
LIN {X 100.418,Y 89.403,Z 81.264,A 180.000,B 0.000,C 180.000} C_DIS
LIN {X 100.346,Y 89.377,Z 81.261,A 180.000,B 0.000,C 180.000} C_DIS
LIN {X 100.199,Y 89.327,Z 81.256,A 180.000,B 0.000,C 180.000} C_DIS
LIN {X 100.125,Y 89.302,Z 81.253,A 180.000,B 0.000,C 180.000} C_DIS
LIN {X 99.977,Y 89.252,Z 81.248,A 180.000,B 0.000,C 180.000} C_DIS
LIN {X 99.903,Y 89.227,Z 81.245,A 180.000,B 0.000,C 180.000} C_DIS
LIN {X 99.829,Y 89.204,Z 81.242,A 180.000,B 0.000,C 180.000} C_DIS
LIN {X 99.755,Y 89.183,Z 81.240,A 180.000,B 0.000,C 180.000} C_DIS
LIN {X 99.530,Y 89.121,Z 81.231,A 180.000,B 0.000,C 180.000} C_DIS
LIN {X 99.456,Y 89.101,Z 81.229,A 180.000,B 0.000,C 180.000} C_DIS
LIN {X 99.380,Y 89.084,Z 81.226,A 180.000,B 0.000,C 180.000} C_DIS
LIN {X 99.305,Y 89.068,Z 81.223,A 180.000,B 0.000,C 180.000} C_DIS
LIN {X 99.152,Y 89.035,Z 81.218,A 180.000,B 0.000,C 180.000} C_DIS
LIN {X 99.075,Y 89.019,Z 81.215,A 180.000,B 0.000,C 180.000} C_DIS
LIN {X 98.998,Y 89.003,Z 81.212,A 180.000,B 0.000,C 180.000} C_DIS
LIN {X 98.922,Y 88.987,Z 81.210,A 180.000,B 0.000,C 180.000} C_DIS
LIN {X 98.845,Y 88.973,Z 81.207,A 180.000,B 0.000,C 180.000} C_DIS
LIN {X 98.769,Y 88.960,Z 81.204,A 180.000,B 0.000,C 180.000} C_DIS
LIN {X 98.692,Y 88.948,Z 81.202,A 180.000,B 0.000,C 180.000} C_DIS
LIN {X 98.615,Y 88.936,Z 81.199,A 180.000,B 0.000,C 180.000} C_DIS
LIN {X 98.538,Y 88.924,Z 81.196,A 180.000,B 0.000,C 180.000} C_DIS
LIN {X 98.461,Y 88.914,Z 81.193,A 180.000,B 0.000,C 180.000} C_DIS
LIN {X 98.384,Y 88.906,Z 81.191,A 180.000,B 0.000,C 180.000} C_DIS
LIN {X 98.229,Y 88.890,Z 81.185,A 180.000,B 0.000,C 180.000} C_DIS
LIN {X 98.151,Y 88.882,Z 81.183,A 180.000,B 0.000,C 180.000} C_DIS
LIN {X 98.073,Y 88.876,Z 81.180,A 180.000,B 0.000,C 180.000} C_DIS
LIN {X 97.995,Y 88.870,Z 81.177,A 180.000,B 0.000,C 180.000} C_DIS
LIN {X 97.917,Y 88.863,Z 81.175,A 180.000,B 0.000,C 180.000} C_DIS
LIN {X 97.840,Y 88.858,Z 81.172,A 180.000,B 0.000,C 180.000} C_DIS
LIN {X 97.762,Y 88.855,Z 81.169,A 180.000,B 0.000,C 180.000} C_DIS
LIN {X 97.683,Y 88.852,Z 81.167,A 180.000,B 0.000,C 180.000} C_DIS
LIN {X 97.605,Y 88.848,Z 81.164,A 180.000,B 0.000,C 180.000} C_DIS
LIN {X 97.527,Y 88.845,Z 81.162,A 180.000,B 0.000,C 180.000} C_DIS
LIN {X 97.448,Y 88.844,Z 81.159,A 180.000,B 0.000,C 180.000} C_DIS
LIN {X 97.370,Y 88.845,Z 81.157,A 180.000,B 0.000,C 180.000} C_DIS
LIN {X 97.292,Y 88.846,Z 81.154,A 180.000,B 0.000,C 180.000} C_DIS
LIN {X 97.137,Y 88.849,Z 81.149,A 180.000,B 0.000,C 180.000} C_DIS
LIN {X 96.981,Y 88.856,Z 81.144,A 180.000,B 0.000,C 180.000} C_DIS
LIN {X 96.825,Y 88.864,Z 81.139,A 180.000,B 0.000,C 180.000} C_DIS
LIN {X 96.669,Y 88.875,Z 81.135,A 180.000,B 0.000,C 180.000} C_DIS
LIN {X 96.513,Y 88.887,Z 81.130,A 180.000,B 0.000,C 180.000} C_DIS
LIN {X 96.357,Y 88.905,Z 81.125,A 180.000,B 0.000,C 180.000} C_DIS
LIN {X 96.202,Y 88.925,Z 81.120,A 180.000,B 0.000,C 180.000} C_DIS
LIN {X 96.047,Y 88.948,Z 81.116,A 180.000,B 0.000,C 180.000} C_DIS
LIN {X 95.893,Y 88.976,Z 81.112,A 180.000,B 0.000,C 180.000} C_DIS
LIN {X 95.739,Y 89.004,Z 81.107,A 180.000,B 0.000,C 180.000} C_DIS
LIN {X 95.585,Y 89.033,Z 81.103,A 180.000,B 0.000,C 180.000} C_DIS
LIN {X 95.432,Y 89.066,Z 81.098,A 180.000,B 0.000,C 180.000} C_DIS
LIN {X 95.280,Y 89.104,Z 81.094,A 180.000,B 0.000,C 180.000} C_DIS
LIN {X 95.128,Y 89.142,Z 81.090,A 180.000,B 0.000,C 180.000} C_DIS
LIN {X 94.978,Y 89.187,Z 81.086,A 180.000,B 0.000,C 180.000} C_DIS
LIN {X 94.828,Y 89.233,Z 81.082,A 180.000,B 0.000,C 180.000} C_DIS
LIN {X 94.678,Y 89.280,Z 81.078,A 180.000,B 0.000,C 180.000} C_DIS
LIN {X 94.529,Y 89.329,Z 81.075,A 180.000,B 0.000,C 180.000} C_DIS
LIN {X 94.382,Y 89.383,Z 81.071,A 180.000,B 0.000,C 180.000} C_DIS
LIN {X 94.235,Y 89.437,Z 81.067,A 180.000,B 0.000,C 180.000} C_DIS
LIN {X 94.090,Y 89.497,Z 81.064,A 180.000,B 0.000,C 180.000} C_DIS
LIN {X 93.946,Y 89.560,Z 81.060,A 180.000,B 0.000,C 180.000} C_DIS
LIN {X 93.803,Y 89.624,Z 81.057,A 180.000,B 0.000,C 180.000} C_DIS
LIN {X 93.660,Y 89.690,Z 81.053,A 180.000,B 0.000,C 180.000} C_DIS
LIN {X 93.519,Y 89.759,Z 81.050,A 180.000,B 0.000,C 180.000} C_DIS
LIN {X 93.379,Y 89.830,Z 81.047,A 180.000,B 0.000,C 180.000} C_DIS
LIN {X 93.240,Y 89.904,Z 81.044,A 180.000,B 0.000,C 180.000} C_DIS
LIN {X 93.104,Y 89.982,Z 81.041,A 180.000,B 0.000,C 180.000} C_DIS
LIN {X 92.968,Y 90.061,Z 81.038,A 180.000,B 0.000,C 180.000} C_DIS
LIN {X 92.834,Y 90.144,Z 81.035,A 180.000,B 0.000,C 180.000} C_DIS
LIN {X 92.702,Y 90.228,Z 81.033,A 180.000,B 0.000,C 180.000} C_DIS
LIN {X 92.570,Y 90.315,Z 81.030,A 180.000,B 0.000,C 180.000} C_DIS
LIN {X 92.439,Y 90.402,Z 81.028,A 180.000,B 0.000,C 180.000} C_DIS
LIN {X 92.186,Y 90.589,Z 81.023,A 180.000,B 0.000,C 180.000} C_DIS
LIN {X 91.940,Y 90.785,Z 81.019,A 180.000,B 0.000,C 180.000} C_DIS
LIN {X 91.699,Y 90.987,Z 81.015,A 180.000,B 0.000,C 180.000} C_DIS
LIN {X 91.467,Y 91.199,Z 81.012,A 180.000,B 0.000,C 180.000} C_DIS
LIN {X 91.244,Y 91.422,Z 81.009,A 180.000,B 0.000,C 180.000} C_DIS
LIN {X 91.027,Y 91.650,Z 81.006,A 180.000,B 0.000,C 180.000} C_DIS
LIN {X 90.819,Y 91.886,Z 81.004,A 180.000,B 0.000,C 180.000} C_DIS
LIN {X 90.620,Y 92.130,Z 81.002,A 180.000,B 0.000,C 180.000} C_DIS
LIN {X 90.431,Y 92.383,Z 81.001,A 180.000,B 0.000,C 180.000} C_DIS
LIN {X 90.250,Y 92.640,Z 81.000,A 180.000,B 0.000,C 180.000} C_DIS
LIN {X 90.082,Y 92.898,Z 81.000,A 180.000,B 0.000,C 180.000} C_DIS
; Cutting Move Starts
LIN {X 90.043,Y 92.964,Z 81.000,A 180.000,B 0.000,C 180.000} C_DIS
LIN {X 89.937,Y 93.142,Z 81.000,A 180.000,B 0.000,C 180.000} C_DIS
LIN {X 89.925,Y 93.165,Z 81.000,A 180.000,B 0.000,C 180.000} C_DIS
LIN {X 89.838,Y 93.321,Z 81.000,A 180.000,B 0.000,C 180.000} C_DIS
LIN {X 89.746,Y 93.495,Z 81.000,A 180.000,B 0.000,C 180.000} C_DIS
LIN {X 89.651,Y 93.679,Z 81.000,A 180.000,B 0.000,C 180.000} C_DIS
LIN {X 89.568,Y 93.857,Z 81.000,A 180.000,B 0.000,C 180.000} C_DIS
LIN {X 89.488,Y 94.036,Z 81.000,A 180.000,B 0.000,C 180.000} C_DIS
LIN {X 89.415,Y 94.215,Z 81.000,A 180.000,B 0.000,C 180.000} C_DIS
LIN {X 89.388,Y 94.282,Z 81.000,A 180.000,B 0.000,C 180.000} C_DIS
LIN {X 89.345,Y 94.394,Z 81.000,A 180.000,B 0.000,C 180.000} C_DIS
LIN {X 89.277,Y 94.573,Z 81.000,A 180.000,B 0.000,C 180.000} C_DIS
LIN {X 89.215,Y 94.751,Z 81.000,A 180.000,B 0.000,C 180.000} C_DIS
LIN {X 89.158,Y 94.930,Z 81.000,A 180.000,B 0.000,C 180.000} C_DIS
LIN {X 89.106,Y 95.109,Z 81.000,A 180.000,B 0.000,C 180.000} C_DIS
LIN {X 89.059,Y 95.288,Z 81.000,A 180.000,B 0.000,C 180.000} C_DIS
LIN {X 89.031,Y 95.399,Z 81.000,A 180.000,B 0.000,C 180.000} C_DIS
LIN {X 89.013,Y 95.466,Z 81.000,A 180.000,B 0.000,C 180.000} C_DIS
LIN {X 88.970,Y 95.645,Z 81.000,A 180.000,B 0.000,C 180.000} C_DIS
LIN {X 88.934,Y 95.824,Z 81.000,A 180.000,B 0.000,C 180.000} C_DIS
LIN {X 88.899,Y 96.003,Z 81.000,A 180.000,B 0.000,C 180.000} C_DIS
LIN {X 88.873,Y 96.181,Z 81.000,A 180.000,B 0.000,C 180.000} C_DIS
LIN {X 88.852,Y 96.330,Z 81.000,A 180.000,B 0.000,C 180.000} C_DIS
LIN {X 88.848,Y 96.360,Z 81.000,A 180.000,B 0.000,C 180.000} C_DIS
LIN {X 88.829,Y 96.510,Z 81.000,A 180.000,B 0.000,C 180.000} C_DIS
LIN {X 88.825,Y 96.539,Z 81.000,A 180.000,B 0.000,C 180.000} C_DIS
LIN {X 88.807,Y 96.718,Z 81.000,A 180.000,B 0.000,C 180.000} C_DIS
LIN {X 88.792,Y 96.897,Z 81.000,A 180.000,B 0.000,C 180.000} C_DIS
LIN {X 88.781,Y 97.075,Z 81.000,A 180.000,B 0.000,C 180.000} C_DIS
LIN {X 88.776,Y 97.254,Z 81.000,A 180.000,B 0.000,C 180.000} C_DIS
LIN {X 88.773,Y 97.433,Z 81.000,A 180.000,B 0.000,C 180.000} C_DIS
LIN {X 88.773,Y 97.612,Z 81.000,A 180.000,B 0.000,C 180.000} C_DIS
LIN {X 88.777,Y 97.790,Z 81.000,A 180.000,B 0.000,C 180.000} C_DIS
LIN {X 88.782,Y 97.969,Z 81.000,A 180.000,B 0.000,C 180.000} C_DIS
LIN {X 88.795,Y 98.148,Z 81.000,A 180.000,B 0.000,C 180.000} C_DIS
LIN {X 88.810,Y 98.327,Z 81.000,A 180.000,B 0.000,C 180.000} C_DIS
LIN {X 88.831,Y 98.505,Z 81.000,A 180.000,B 0.000,C 180.000} C_DIS
LIN {X 88.852,Y 98.670,Z 81.000,A 180.000,B 0.000,C 180.000} C_DIS
LIN {X 88.879,Y 98.863,Z 81.000,A 180.000,B 0.000,C 180.000} C_DIS
LIN {X 88.907,Y 99.042,Z 81.000,A 180.000,B 0.000,C 180.000} C_DIS
LIN {X 88.943,Y 99.221,Z 81.000,A 180.000,B 0.000,C 180.000} C_DIS
LIN {X 88.980,Y 99.399,Z 81.000,A 180.000,B 0.000,C 180.000} C_DIS
LIN {X 89.025,Y 99.578,Z 81.000,A 180.000,B 0.000,C 180.000} C_DIS
LIN {X 89.031,Y 99.601,Z 81.000,A 180.000,B 0.000,C 180.000} C_DIS
LIN {X 89.071,Y 99.757,Z 81.000,A 180.000,B 0.000,C 180.000} C_DIS
LIN {X 89.117,Y 99.936,Z 81.000,A 180.000,B 0.000,C 180.000} C_DIS
LIN {X 89.172,Y 100.114,Z 81.000,A 180.000,B 0.000,C 180.000} C_DIS
LIN {X 89.209,Y 100.232,Z 81.000,A 180.000,B 0.000,C 180.000} C_DIS
LIN {X 89.229,Y 100.293,Z 81.000,A 180.000,B 0.000,C 180.000} C_DIS
LIN {X 89.294,Y 100.472,Z 81.000,A 180.000,B 0.000,C 180.000} C_DIS
LIN {X 89.362,Y 100.651,Z 81.000,A 180.000,B 0.000,C 180.000} C_DIS
LIN {X 89.388,Y 100.718,Z 81.000,A 180.000,B 0.000,C 180.000} C_DIS
LIN {X 89.432,Y 100.829,Z 81.000,A 180.000,B 0.000,C 180.000} C_DIS
LIN {X 89.507,Y 101.008,Z 81.000,A 180.000,B 0.000,C 180.000} C_DIS
LIN {X 89.587,Y 101.187,Z 81.000,A 180.000,B 0.000,C 180.000} C_DIS
LIN {X 89.674,Y 101.366,Z 81.000,A 180.000,B 0.000,C 180.000} C_DIS
LIN {X 89.766,Y 101.545,Z 81.000,A 180.000,B 0.000,C 180.000} C_DIS
LIN {X 89.863,Y 101.723,Z 81.000,A 180.000,B 0.000,C 180.000} C_DIS
LIN {X 89.925,Y 101.835,Z 81.000,A 180.000,B 0.000,C 180.000} C_DIS
LIN {X 89.964,Y 101.902,Z 81.000,A 180.000,B 0.000,C 180.000} C_DIS
LIN {X 90.069,Y 102.081,Z 81.000,A 180.000,B 0.000,C 180.000} C_DIS
LIN {X 90.103,Y 102.138,Z 81.000,A 180.000,B 0.000,C 180.000} C_DIS
LIN {X 90.183,Y 102.260,Z 81.000,A 180.000,B 0.000,C 180.000} C_DIS
LIN {X 90.282,Y 102.408,Z 81.000,A 180.000,B 0.000,C 180.000} C_DIS
LIN {X 90.302,Y 102.438,Z 81.000,A 180.000,B 0.000,C 180.000} C_DIS
LIN {X 90.431,Y 102.617,Z 81.000,A 180.000,B 0.000,C 180.000} C_DIS
LIN {X 90.461,Y 102.659,Z 81.000,A 180.000,B 0.000,C 180.000} C_DIS
LIN {X 90.563,Y 102.796,Z 81.000,A 180.000,B 0.000,C 180.000} C_DIS
LIN {X 90.640,Y 102.897,Z 81.000,A 180.000,B 0.000,C 180.000} C_DIS
LIN {X 90.700,Y 102.975,Z 81.000,A 180.000,B 0.000,C 180.000} C_DIS
LIN {X 90.818,Y 103.116,Z 81.000,A 180.000,B 0.000,C 180.000} C_DIS
LIN {X 90.850,Y 103.153,Z 81.000,A 180.000,B 0.000,C 180.000} C_DIS
LIN {X 90.997,Y 103.322,Z 81.000,A 180.000,B 0.000,C 180.000} C_DIS
LIN {X 91.007,Y 103.332,Z 81.000,A 180.000,B 0.000,C 180.000} C_DIS
LIN {X 91.176,Y 103.512,Z 81.000,A 180.000,B 0.000,C 180.000} C_DIS
LIN {X 91.344,Y 103.690,Z 81.000,A 180.000,B 0.000,C 180.000} C_DIS
LIN {X 91.355,Y 103.700,Z 81.000,A 180.000,B 0.000,C 180.000} C_DIS
LIN {X 91.531,Y 103.869,Z 81.000,A 180.000,B 0.000,C 180.000} C_DIS
LIN {X 91.533,Y 103.871,Z 81.000,A 180.000,B 0.000,C 180.000} C_DIS
LIN {X 91.712,Y 104.034,Z 81.000,A 180.000,B 0.000,C 180.000} C_DIS
LIN {X 91.891,Y 104.185,Z 81.000,A 180.000,B 0.000,C 180.000} C_DIS
LIN {X 91.940,Y 104.226,Z 81.000,A 180.000,B 0.000,C 180.000} C_DIS
LIN {X 92.070,Y 104.333,Z 81.000,A 180.000,B 0.000,C 180.000} C_DIS
LIN {X 92.160,Y 104.405,Z 81.000,A 180.000,B 0.000,C 180.000} C_DIS
LIN {X 92.249,Y 104.472,Z 81.000,A 180.000,B 0.000,C 180.000} C_DIS
LIN {X 92.397,Y 104.584,Z 81.000,A 180.000,B 0.000,C 180.000} C_DIS
LIN {X 92.427,Y 104.605,Z 81.000,A 180.000,B 0.000,C 180.000} C_DIS
LIN {X 92.606,Y 104.726,Z 81.000,A 180.000,B 0.000,C 180.000} C_DIS
LIN {X 92.660,Y 104.762,Z 81.000,A 180.000,B 0.000,C 180.000} C_DIS
LIN {X 92.785,Y 104.844,Z 81.000,A 180.000,B 0.000,C 180.000} C_DIS
LIN {X 92.938,Y 104.941,Z 81.000,A 180.000,B 0.000,C 180.000} C_DIS
LIN {X 92.964,Y 104.957,Z 81.000,A 180.000,B 0.000,C 180.000} C_DIS
LIN {X 93.142,Y 105.063,Z 81.000,A 180.000,B 0.000,C 180.000} C_DIS
LIN {X 93.240,Y 105.120,Z 81.000,A 180.000,B 0.000,C 180.000} C_DIS
LIN {X 93.321,Y 105.165,Z 81.000,A 180.000,B 0.000,C 180.000} C_DIS
LIN {X 93.500,Y 105.258,Z 81.000,A 180.000,B 0.000,C 180.000} C_DIS
LIN {X 93.580,Y 105.299,Z 81.000,A 180.000,B 0.000,C 180.000} C_DIS
LIN {X 93.679,Y 105.347,Z 81.000,A 180.000,B 0.000,C 180.000} C_DIS
LIN {X 93.857,Y 105.431,Z 81.000,A 180.000,B 0.000,C 180.000} C_DIS
LIN {X 93.961,Y 105.477,Z 81.000,A 180.000,B 0.000,C 180.000} C_DIS
LIN {X 94.036,Y 105.511,Z 81.000,A 180.000,B 0.000,C 180.000} C_DIS
LIN {X 94.215,Y 105.589,Z 81.000,A 180.000,B 0.000,C 180.000} C_DIS
LIN {X 94.394,Y 105.657,Z 81.000,A 180.000,B 0.000,C 180.000} C_DIS
LIN {X 94.573,Y 105.724,Z 81.000,A 180.000,B 0.000,C 180.000} C_DIS
LIN {X 94.751,Y 105.782,Z 81.000,A 180.000,B 0.000,C 180.000} C_DIS
LIN {X 94.916,Y 105.835,Z 81.000,A 180.000,B 0.000,C 180.000} C_DIS
LIN {X 94.930,Y 105.839,Z 81.000,A 180.000,B 0.000,C 180.000} C_DIS
LIN {X 95.109,Y 105.896,Z 81.000,A 180.000,B 0.000,C 180.000} C_DIS
LIN {X 95.288,Y 105.944,Z 81.000,A 180.000,B 0.000,C 180.000} C_DIS
LIN {X 95.466,Y 105.990,Z 81.000,A 180.000,B 0.000,C 180.000} C_DIS
LIN {X 95.573,Y 106.014,Z 81.000,A 180.000,B 0.000,C 180.000} C_DIS
LIN {X 95.645,Y 106.028,Z 81.000,A 180.000,B 0.000,C 180.000} C_DIS
LIN {X 95.824,Y 106.064,Z 81.000,A 180.000,B 0.000,C 180.000} C_DIS
LIN {X 96.003,Y 106.098,Z 81.000,A 180.000,B 0.000,C 180.000} C_DIS
LIN {X 96.181,Y 106.129,Z 81.000,A 180.000,B 0.000,C 180.000} C_DIS
LIN {X 96.360,Y 106.154,Z 81.000,A 180.000,B 0.000,C 180.000} C_DIS
LIN {X 96.539,Y 106.177,Z 81.000,A 180.000,B 0.000,C 180.000} C_DIS
LIN {X 96.721,Y 106.193,Z 81.000,A 180.000,B 0.000,C 180.000} C_DIS
LIN {X 96.897,Y 106.207,Z 81.000,A 180.000,B 0.000,C 180.000} C_DIS
LIN {X 97.075,Y 106.218,Z 81.000,A 180.000,B 0.000,C 180.000} C_DIS
LIN {X 97.254,Y 106.225,Z 81.000,A 180.000,B 0.000,C 180.000} C_DIS
LIN {X 97.433,Y 106.230,Z 81.000,A 180.000,B 0.000,C 180.000} C_DIS
LIN {X 97.612,Y 106.228,Z 81.000,A 180.000,B 0.000,C 180.000} C_DIS
LIN {X 97.790,Y 106.223,Z 81.000,A 180.000,B 0.000,C 180.000} C_DIS
LIN {X 97.969,Y 106.215,Z 81.000,A 180.000,B 0.000,C 180.000} C_DIS
LIN {X 98.148,Y 106.204,Z 81.000,A 180.000,B 0.000,C 180.000} C_DIS
LIN {X 98.279,Y 106.193,Z 81.000,A 180.000,B 0.000,C 180.000} C_DIS
LIN {X 98.327,Y 106.189,Z 81.000,A 180.000,B 0.000,C 180.000} C_DIS
LIN {X 98.505,Y 106.172,Z 81.000,A 180.000,B 0.000,C 180.000} C_DIS
LIN {X 98.684,Y 106.148,Z 81.000,A 180.000,B 0.000,C 180.000} C_DIS
LIN {X 98.863,Y 106.122,Z 81.000,A 180.000,B 0.000,C 180.000} C_DIS
LIN {X 99.042,Y 106.090,Z 81.000,A 180.000,B 0.000,C 180.000} C_DIS
LIN {X 99.221,Y 106.055,Z 81.000,A 180.000,B 0.000,C 180.000} C_DIS
LIN {X 99.399,Y 106.019,Z 81.000,A 180.000,B 0.000,C 180.000} C_DIS
LIN {X 99.427,Y 106.014,Z 81.000,A 180.000,B 0.000,C 180.000} C_DIS
LIN {X 99.578,Y 105.978,Z 81.000,A 180.000,B 0.000,C 180.000} C_DIS
LIN {X 99.757,Y 105.932,Z 81.000,A 180.000,B 0.000,C 180.000} C_DIS
LIN {X 99.936,Y 105.882,Z 81.000,A 180.000,B 0.000,C 180.000} C_DIS
LIN {X 100.114,Y 105.825,Z 81.000,A 180.000,B 0.000,C 180.000} C_DIS
LIN {X 100.293,Y 105.768,Z 81.000,A 180.000,B 0.000,C 180.000} C_DIS
LIN {X 100.472,Y 105.708,Z 81.000,A 180.000,B 0.000,C 180.000} C_DIS
LIN {X 100.608,Y 105.656,Z 81.000,A 180.000,B 0.000,C 180.000} C_DIS
LIN {X 100.651,Y 105.640,Z 81.000,A 180.000,B 0.000,C 180.000} C_DIS
LIN {X 100.829,Y 105.570,Z 81.000,A 180.000,B 0.000,C 180.000} C_DIS
LIN {X 101.008,Y 105.491,Z 81.000,A 180.000,B 0.000,C 180.000} C_DIS
LIN {X 101.039,Y 105.477,Z 81.000,A 180.000,B 0.000,C 180.000} C_DIS
LIN {X 101.187,Y 105.410,Z 81.000,A 180.000,B 0.000,C 180.000} C_DIS
LIN {X 101.366,Y 105.326,Z 81.000,A 180.000,B 0.000,C 180.000} C_DIS
LIN {X 101.420,Y 105.299,Z 81.000,A 180.000,B 0.000,C 180.000} C_DIS
LIN {X 101.545,Y 105.235,Z 81.000,A 180.000,B 0.000,C 180.000} C_DIS
LIN {X 101.723,Y 105.141,Z 81.000,A 180.000,B 0.000,C 180.000} C_DIS
LIN {X 101.760,Y 105.120,Z 81.000,A 180.000,B 0.000,C 180.000} C_DIS
LIN {X 101.902,Y 105.037,Z 81.000,A 180.000,B 0.000,C 180.000} C_DIS
LIN {X 102.062,Y 104.941,Z 81.000,A 180.000,B 0.000,C 180.000} C_DIS
LIN {X 102.081,Y 104.929,Z 81.000,A 180.000,B 0.000,C 180.000} C_DIS
LIN {X 102.260,Y 104.816,Z 81.000,A 180.000,B 0.000,C 180.000} C_DIS
LIN {X 102.340,Y 104.762,Z 81.000,A 180.000,B 0.000,C 180.000} C_DIS
LIN {X 102.438,Y 104.697,Z 81.000,A 180.000,B 0.000,C 180.000} C_DIS
LIN {X 102.603,Y 104.584,Z 81.000,A 180.000,B 0.000,C 180.000} C_DIS
LIN {X 102.617,Y 104.573,Z 81.000,A 180.000,B 0.000,C 180.000} C_DIS
LIN {X 102.796,Y 104.438,Z 81.000,A 180.000,B 0.000,C 180.000} C_DIS
LIN {X 102.840,Y 104.405,Z 81.000,A 180.000,B 0.000,C 180.000} C_DIS
LIN {X 102.975,Y 104.297,Z 81.000,A 180.000,B 0.000,C 180.000} C_DIS
LIN {X 103.060,Y 104.226,Z 81.000,A 180.000,B 0.000,C 180.000} C_DIS
LIN {X 103.153,Y 104.148,Z 81.000,A 180.000,B 0.000,C 180.000} C_DIS
LIN {X 103.272,Y 104.047,Z 81.000,A 180.000,B 0.000,C 180.000} C_DIS
LIN {X 103.332,Y 103.996,Z 81.000,A 180.000,B 0.000,C 180.000} C_DIS
LIN {X 103.469,Y 103.869,Z 81.000,A 180.000,B 0.000,C 180.000} C_DIS
LIN {X 103.511,Y 103.829,Z 81.000,A 180.000,B 0.000,C 180.000} C_DIS
LIN {X 103.656,Y 103.690,Z 81.000,A 180.000,B 0.000,C 180.000} C_DIS
LIN {X 103.690,Y 103.654,Z 81.000,A 180.000,B 0.000,C 180.000} C_DIS
LIN {X 103.869,Y 103.465,Z 81.000,A 180.000,B 0.000,C 180.000} C_DIS
LIN {X 103.993,Y 103.332,Z 81.000,A 180.000,B 0.000,C 180.000} C_DIS
LIN {X 104.047,Y 103.274,Z 81.000,A 180.000,B 0.000,C 180.000} C_DIS
LIN {X 104.150,Y 103.153,Z 81.000,A 180.000,B 0.000,C 180.000} C_DIS
LIN {X 104.226,Y 103.064,Z 81.000,A 180.000,B 0.000,C 180.000} C_DIS
LIN {X 104.300,Y 102.975,Z 81.000,A 180.000,B 0.000,C 180.000} C_DIS
LIN {X 104.405,Y 102.838,Z 81.000,A 180.000,B 0.000,C 180.000} C_DIS
LIN {X 104.437,Y 102.796,Z 81.000,A 180.000,B 0.000,C 180.000} C_DIS
LIN {X 104.569,Y 102.617,Z 81.000,A 180.000,B 0.000,C 180.000} C_DIS
